// TwinCAT 3 PLC project SIM_1
// ProgramVersion: 3.1.4026.25
// libraries:
//   OC_Core, * (Open Commissioning)
//   OC_EtherCAT, * (Open Commissioning)
//   Tc2_Math, * (Beckhoff Automation GmbH)
//   Tc2_Standard, * (Beckhoff Automation GmbH)
//   Tc2_System, * (Beckhoff Automation GmbH)
//   Tc2_Utilities, * (Beckhoff Automation GmbH)
//   Tc3_Module, * (Beckhoff Automation GmbH)
// project tree:
//   Hil/EtherCAT_1_SIM/ GVL_EtherCAT_1_SIM.TcGVL, PRG_EtherCAT_1_SIM.TcPOU
//   Library/ FB_Camera.TcPOU (not stored)
//   FG_01/ FG_01.TcPOU
//   FG_02/ FG_02.TcPOU
//   FG_03/ FG_03.TcPOU
//   FG_04/ FG_04.TcPOU
//   FG_05/ FG_05.TcPOU
//   FG_System/ FG_System.TcPOU
//   FG_Transport/ FG_Transport.TcPOU
//   / MAIN.TcPOU, PlcTask.TcTTO (not stored)
// real-time tasks:
//   TASK PlcTask_SIM: cycle T#1ms, priority 4, ADS port 350
//   TASK PlcTask_PLC: cycle T#10ms, priority 20, ADS port 351
// I/O:
//   DEVICE EtherCAT_1_SIM, AmsNetId 169.254.215.222.4.1
//     FG_System_EK1100 // EK1100-0000-0018
//     FG_System_Panel_EL1809_1 // EL1809-0000-0018
//     FG_System_Panel_EL2809_1 // EL2809-0000-0018
//     FG_System_Door_EL1809_1 // EL1809-0000-0018
//     FG_System_Door_EL2008_1 // EL2008-0000-0018
//     FG_Transport_EK1100 // EK1100-0000-0018
//     FG_Transport_Index_EL1809_1 // EL1809-0000-0018
//     FG_Transport_Index_EL1809_2 // EL1809-0000-0018
//     FG_Transport_Stopper_EL1809_1 // EL1809-0000-0018
//     FG_Transport_Lift_EL1809_1 // EL1809-0000-0018
//     FG_Transport_Drive_EL1008_1 // EL1008-0000-0018
//     FG_Transport_Index_EL2809_1 // EL2809-0000-0018
//     FG_Transport_Stopper_EL2008_1 // EL2008-0000-0018
//     FG_Transport_Lift_EL2008_1 // EL2008-0000-0018
//     FG_Transport_Drive_EL2008_1 // EL2008-0000-0018
//     FG_01_EK1100 // EK1100-0000-0018
//     FG_01_EL1008_1 // EL1008-0000-0018
//     FG_01_EL1008_2 // EL1008-0000-0018
//     FG_01_EL2008_1 // EL2008-0000-0018
//     FG_01_EL1859_1 // EL1859-0000-0018
//     FG_01_EL1859_2 // EL1859-0000-0018
//     FG_02_EK1100 // EK1100-0000-0018
//     FG_02_EL1859_1 // EL1859-0000-0018
//     FG_03_EK1100 // EK1100-0000-0018
//     FG_03_EL1809_1 // EL1809-0000-0018
//     FG_03_EL2809_1 // EL2809-0000-0018
//     FG_04_EK1100 // EK1100-0000-0018
//     FG_04_EL1008_1 // EL1008-0000-0018
//     FG_04_EL2008_1 // EL2008-0000-0018
//     FG_05_EK1100 // EK1100-0000-0018
//     FG_05_EL1809_1 // EL1809-0000-0018
//     FG_05_EL2809_1 // EL2809-0000-0018
//     FG_05_EL1859_1 // EL1859-0000-0018
//     FG_05_EL1859_2 // EL1859-0000-0018
//   DEVICE EtherCAT_1, AmsNetId 169.254.215.222.3.1
//     FG_System_EK1100 [EK1100 EtherCAT Coupler (2A E-Bus)]
//       FG_System_Panel_EL1809_1 [EL1809 16Ch. Dig. Input 24V, 3ms]
//       FG_System_Panel_EL2809_1 [EL2809 16Ch. Dig. Output 24V, 0.5A]
//       FG_System_Door_EL1809_1 [EL1809 16Ch. Dig. Input 24V, 3ms]
//       FG_System_Door_EL2008_1 [EL2008 8Ch. Dig. Output 24V, 0.5A]
//     FG_Transport_EK1100 [EK1100 EtherCAT Coupler (2A E-Bus)]
//       FG_Transport_Index_EL1809_1 [EL1809 16Ch. Dig. Input 24V, 3ms]
//       FG_Transport_Index_EL1809_2 [EL1809 16Ch. Dig. Input 24V, 3ms]
//       FG_Transport_Stopper_EL1809_1 [EL1809 16Ch. Dig. Input 24V, 3ms]
//       FG_Transport_Lift_EL1809_1 [EL1809 16Ch. Dig. Input 24V, 3ms]
//       FG_Transport_Drive_EL1008_1 [EL1008 8Ch. Dig. Input 24V, 3ms]
//       FG_Transport_Index_EL2809_1 [EL2809 16Ch. Dig. Output 24V, 0.5A]
//       FG_Transport_Stopper_EL2008_1 [EL2008 8Ch. Dig. Output 24V, 0.5A]
//       FG_Transport_Lift_EL2008_1 [EL2008 8Ch. Dig. Output 24V, 0.5A]
//       FG_Transport_Drive_EL2008_1 [EL2008 8Ch. Dig. Output 24V, 0.5A]
//     FG_01_EK1100 [EK1100 EtherCAT Coupler (2A E-Bus)]
//       FG_01_EL1008_1 [EL1008 8Ch. Dig. Input 24V, 3ms]
//       FG_01_EL1008_2 [EL1008 8Ch. Dig. Input 24V, 3ms]
//       FG_01_EL2008_1 [EL2008 8Ch. Dig. Output 24V, 0.5A]
//       FG_01_EL1859_1 [EL1859 8Ch. Dig. Input 24V, 3ms, 8Ch. Dig. Output 24V, 0.5A]
//       FG_01_EL1859_2 [EL1859 8Ch. Dig. Input 24V, 3ms, 8Ch. Dig. Output 24V, 0.5A]
//     FG_02_EK1100 [EK1100 EtherCAT Coupler (2A E-Bus)]
//       FG_02_EL1859_1 [EL1859 8Ch. Dig. Input 24V, 3ms, 8Ch. Dig. Output 24V, 0.5A]
//     FG_03_EK1100 [EK1100 EtherCAT Coupler (2A E-Bus)]
//       FG_03_EL1809_1 [EL1809 16Ch. Dig. Input 24V, 3ms]
//       FG_03_EL2809_1 [EL2809 16Ch. Dig. Output 24V, 0.5A]
//     FG_04_EK1100 [EK1100 EtherCAT Coupler (2A E-Bus)]
//       FG_04_EL1008_1 [EL1008 8Ch. Dig. Input 24V, 3ms]
//       FG_04_EL2008_1 [EL2008 8Ch. Dig. Output 24V, 0.5A]
//     FG_05_EK1100 [EK1100 EtherCAT Coupler (2A E-Bus)]
//       FG_05_EL1809_1 [EL1809 16Ch. Dig. Input 24V, 3ms]
//       FG_05_EL2809_1 [EL2809 16Ch. Dig. Output 24V, 0.5A]
//       FG_05_EL1859_1 [EL1859 8Ch. Dig. Input 24V, 3ms, 8Ch. Dig. Output 24V, 0.5A]
//       FG_05_EL1859_2 [EL1859 8Ch. Dig. Input 24V, 3ms, 8Ch. Dig. Output 24V, 0.5A]
// variable links:
//   PLC_1/PLC_1 Instance <-> EtherCAT_1/FG_01_EK1100/FG_01_EL1008_1
//     PlcTask Inputs/MAIN.Machine.FG_01.Y_Gripper.ExtendedSensor <-> Channel 2/Input
//     PlcTask Inputs/MAIN.Machine.FG_01.Y_Gripper.RetractedSensor <-> Channel 1/Input
//     PlcTask Inputs/MAIN.Machine.FG_01.Y_Platform.ExtendedSensor <-> Channel 4/Input
//     PlcTask Inputs/MAIN.Machine.FG_01.Y_Platform.RetractedSensor <-> Channel 3/Input
//     PlcTask Inputs/MAIN.Machine.FG_01.Y_ReaderWindow.ExtendedSensor <-> Channel 6/Input
//     PlcTask Inputs/MAIN.Machine.FG_01.Y_ReaderWindow.RetractedSensor <-> Channel 5/Input
//   PLC_1/PLC_1 Instance <-> EtherCAT_1/FG_01_EK1100/FG_01_EL1008_2
//     PlcTask Inputs/MAIN.Machine.FG_01.B_SafetyGate1.HardwareInput <-> Channel 5/Input
//     PlcTask Inputs/MAIN.Machine.FG_01.B_SafetyGate2.HardwareInput <-> Channel 6/Input
//     PlcTask Inputs/MAIN.Machine.FG_01.Y_Gate1.ExtendedSensor <-> Channel 2/Input
//     PlcTask Inputs/MAIN.Machine.FG_01.Y_Gate2.ExtendedSensor <-> Channel 4/Input
//     PlcTask Inputs/MAIN.Machine.FG_01.Y_Gate1.RetractedSensor <-> Channel 1/Input
//     PlcTask Inputs/MAIN.Machine.FG_01.Y_Gate2.RetractedSensor <-> Channel 3/Input
//   PLC_1/PLC_1 Instance <-> EtherCAT_1/FG_01_EK1100/FG_01_EL1859_1
//     PlcTask Inputs/MAIN.Machine.FG_01.P_Camera.InputData <-> Channel 1/Input
//     PlcTask Inputs/MAIN.Machine.FG_01.P_Camera.InputData @bit 1 <-> Channel 2/Input
//     PlcTask Inputs/MAIN.Machine.FG_01.P_Camera.InputData @bit 2 <-> Channel 3/Input
//     PlcTask Inputs/MAIN.Machine.FG_01.P_Camera.InputData @bit 3 <-> Channel 4/Input
//     PlcTask Inputs/MAIN.Machine.FG_01.P_Camera.InputData @bit 4 <-> Channel 5/Input
//     PlcTask Inputs/MAIN.Machine.FG_01.P_Camera.InputData @bit 5 <-> Channel 6/Input
//     PlcTask Inputs/MAIN.Machine.FG_01.P_Camera.InputData @bit 6 <-> Channel 7/Input
//     PlcTask Inputs/MAIN.Machine.FG_01.P_Camera.InputData @bit 7 <-> Channel 8/Input
//     PlcTask Outputs/MAIN.Machine.FG_01.P_Camera.OutputData @bit 1 <-> Channel 10/Output
//     PlcTask Outputs/MAIN.Machine.FG_01.P_Camera.OutputData @bit 2 <-> Channel 11/Output
//     PlcTask Outputs/MAIN.Machine.FG_01.P_Camera.OutputData @bit 3 <-> Channel 12/Output
//     PlcTask Outputs/MAIN.Machine.FG_01.P_Camera.OutputData @bit 4 <-> Channel 13/Output
//     PlcTask Outputs/MAIN.Machine.FG_01.P_Camera.OutputData @bit 5 <-> Channel 14/Output
//     PlcTask Outputs/MAIN.Machine.FG_01.P_Camera.OutputData @bit 6 <-> Channel 15/Output
//     PlcTask Outputs/MAIN.Machine.FG_01.P_Camera.OutputData @bit 7 <-> Channel 16/Output
//     PlcTask Outputs/MAIN.Machine.FG_01.P_Camera.OutputData <-> Channel 9/Output
//   PLC_1/PLC_1 Instance <-> EtherCAT_1/FG_01_EK1100/FG_01_EL1859_2
//     PlcTask Inputs/MAIN.Machine.FG_01.Y_LaserMark.InputData <-> Channel 1/Input
//     PlcTask Inputs/MAIN.Machine.FG_01.Y_LaserMark.InputData @bit 1 <-> Channel 2/Input
//     PlcTask Inputs/MAIN.Machine.FG_01.Y_LaserMark.InputData @bit 2 <-> Channel 3/Input
//     PlcTask Inputs/MAIN.Machine.FG_01.Y_LaserMark.InputData @bit 3 <-> Channel 4/Input
//     PlcTask Inputs/MAIN.Machine.FG_01.Y_LaserMark.InputData @bit 4 <-> Channel 5/Input
//     PlcTask Inputs/MAIN.Machine.FG_01.Y_LaserMark.InputData @bit 5 <-> Channel 6/Input
//     PlcTask Inputs/MAIN.Machine.FG_01.Y_LaserMark.InputData @bit 6 <-> Channel 7/Input
//     PlcTask Inputs/MAIN.Machine.FG_01.Y_LaserMark.InputData @bit 7 <-> Channel 8/Input
//     PlcTask Outputs/MAIN.Machine.FG_01.Y_LaserMark.OutputData @bit 1 <-> Channel 10/Output
//     PlcTask Outputs/MAIN.Machine.FG_01.Y_LaserMark.OutputData @bit 2 <-> Channel 11/Output
//     PlcTask Outputs/MAIN.Machine.FG_01.Y_LaserMark.OutputData @bit 3 <-> Channel 12/Output
//     PlcTask Outputs/MAIN.Machine.FG_01.Y_LaserMark.OutputData @bit 4 <-> Channel 13/Output
//     PlcTask Outputs/MAIN.Machine.FG_01.Y_LaserMark.OutputData @bit 5 <-> Channel 14/Output
//     PlcTask Outputs/MAIN.Machine.FG_01.Y_LaserMark.OutputData @bit 6 <-> Channel 15/Output
//     PlcTask Outputs/MAIN.Machine.FG_01.Y_LaserMark.OutputData @bit 7 <-> Channel 16/Output
//     PlcTask Outputs/MAIN.Machine.FG_01.Y_LaserMark.OutputData <-> Channel 9/Output
//   PLC_1/PLC_1 Instance <-> EtherCAT_1/FG_01_EK1100/FG_01_EL2008_1
//     PlcTask Outputs/MAIN.Machine.FG_01.Y_Gate1._ExtendOutput <-> Channel 7/Output
//     PlcTask Outputs/MAIN.Machine.FG_01.Y_Gate2._ExtendOutput <-> Channel 8/Output
//     PlcTask Outputs/MAIN.Machine.FG_01.Y_Gripper._ExtendOutput <-> Channel 1/Output
//     PlcTask Outputs/MAIN.Machine.FG_01.Y_Gripper._RetractOutput <-> Channel 5/Output
//     PlcTask Outputs/MAIN.Machine.FG_01.Y_Platform._ExtendOutput <-> Channel 2/Output
//     PlcTask Outputs/MAIN.Machine.FG_01.Y_Platform._RetractOutput <-> Channel 3/Output
//     PlcTask Outputs/MAIN.Machine.FG_01.Y_ReaderWindow._ExtendOutput <-> Channel 4/Output
//     PlcTask Outputs/MAIN.Machine.FG_01.Y_ReaderWindow._RetractOutput <-> Channel 6/Output
//   PLC_1/PLC_1 Instance <-> EtherCAT_1/FG_02_EK1100/FG_02_EL1859_1
//     PlcTask Inputs/MAIN.Machine.FG_02.P_Camera.InputData <-> Channel 1/Input
//     PlcTask Inputs/MAIN.Machine.FG_02.P_Camera.InputData @bit 1 <-> Channel 2/Input
//     PlcTask Inputs/MAIN.Machine.FG_02.P_Camera.InputData @bit 2 <-> Channel 3/Input
//     PlcTask Inputs/MAIN.Machine.FG_02.P_Camera.InputData @bit 3 <-> Channel 4/Input
//     PlcTask Inputs/MAIN.Machine.FG_02.P_Camera.InputData @bit 4 <-> Channel 5/Input
//     PlcTask Inputs/MAIN.Machine.FG_02.P_Camera.InputData @bit 5 <-> Channel 6/Input
//     PlcTask Inputs/MAIN.Machine.FG_02.P_Camera.InputData @bit 6 <-> Channel 7/Input
//     PlcTask Inputs/MAIN.Machine.FG_02.P_Camera.InputData @bit 7 <-> Channel 8/Input
//     PlcTask Outputs/MAIN.Machine.FG_02.P_Camera.OutputData @bit 1 <-> Channel 10/Output
//     PlcTask Outputs/MAIN.Machine.FG_02.P_Camera.OutputData @bit 2 <-> Channel 11/Output
//     PlcTask Outputs/MAIN.Machine.FG_02.P_Camera.OutputData @bit 3 <-> Channel 12/Output
//     PlcTask Outputs/MAIN.Machine.FG_02.P_Camera.OutputData @bit 4 <-> Channel 13/Output
//     PlcTask Outputs/MAIN.Machine.FG_02.P_Camera.OutputData @bit 5 <-> Channel 14/Output
//     PlcTask Outputs/MAIN.Machine.FG_02.P_Camera.OutputData @bit 6 <-> Channel 15/Output
//     PlcTask Outputs/MAIN.Machine.FG_02.P_Camera.OutputData @bit 7 <-> Channel 16/Output
//     PlcTask Outputs/MAIN.Machine.FG_02.P_Camera.OutputData <-> Channel 9/Output
//   PLC_1/PLC_1 Instance <-> EtherCAT_1/FG_03_EK1100/FG_03_EL1809_1
//     PlcTask Inputs/MAIN.Machine.FG_03.B_Detect1.HardwareInput <-> Channel 15/Input
//     PlcTask Inputs/MAIN.Machine.FG_03.B_Detect2.HardwareInput <-> Channel 16/Input
//     PlcTask Inputs/MAIN.Machine.FG_03.Y_AxisR1.ExtendedSensor <-> Channel 5/Input
//     PlcTask Inputs/MAIN.Machine.FG_03.Y_AxisR1.RetractedSensor <-> Channel 6/Input
//     PlcTask Inputs/MAIN.Machine.FG_03.Y_AxisX1.ExtendedSensor <-> Channel 1/Input
//     PlcTask Inputs/MAIN.Machine.FG_03.Y_AxisX2.ExtendedSensor <-> Channel 9/Input
//     PlcTask Inputs/MAIN.Machine.FG_03.Y_AxisX1.RetractedSensor <-> Channel 2/Input
//     PlcTask Inputs/MAIN.Machine.FG_03.Y_AxisX2.RetractedSensor <-> Channel 10/Input
//     PlcTask Inputs/MAIN.Machine.FG_03.Y_AxisY1.ExtendedSensor <-> Channel 3/Input
//     PlcTask Inputs/MAIN.Machine.FG_03.Y_AxisY2.ExtendedSensor <-> Channel 11/Input
//     PlcTask Inputs/MAIN.Machine.FG_03.Y_AxisY1.RetractedSensor <-> Channel 4/Input
//     PlcTask Inputs/MAIN.Machine.FG_03.Y_AxisY2.RetractedSensor <-> Channel 12/Input
//     PlcTask Inputs/MAIN.Machine.FG_03.Y_Gripper1.ExtendedSensor <-> Channel 7/Input
//     PlcTask Inputs/MAIN.Machine.FG_03.Y_Gripper2.ExtendedSensor <-> Channel 13/Input
//     PlcTask Inputs/MAIN.Machine.FG_03.Y_Gripper1.RetractedSensor <-> Channel 8/Input
//     PlcTask Inputs/MAIN.Machine.FG_03.Y_Gripper2.RetractedSensor <-> Channel 14/Input
//   PLC_1/PLC_1 Instance <-> EtherCAT_1/FG_03_EK1100/FG_03_EL2809_1
//     PlcTask Outputs/MAIN.Machine.FG_03.Y_AxisR1._ExtendOutput <-> Channel 5/Output
//     PlcTask Outputs/MAIN.Machine.FG_03.Y_AxisR1._RetractOutput <-> Channel 6/Output
//     PlcTask Outputs/MAIN.Machine.FG_03.Y_AxisX1._ExtendOutput <-> Channel 1/Output
//     PlcTask Outputs/MAIN.Machine.FG_03.Y_AxisX2._ExtendOutput <-> Channel 9/Output
//     PlcTask Outputs/MAIN.Machine.FG_03.Y_AxisX1._RetractOutput <-> Channel 2/Output
//     PlcTask Outputs/MAIN.Machine.FG_03.Y_AxisX2._RetractOutput <-> Channel 10/Output
//     PlcTask Outputs/MAIN.Machine.FG_03.Y_AxisY1._ExtendOutput <-> Channel 3/Output
//     PlcTask Outputs/MAIN.Machine.FG_03.Y_AxisY2._ExtendOutput <-> Channel 11/Output
//     PlcTask Outputs/MAIN.Machine.FG_03.Y_AxisY1._RetractOutput <-> Channel 4/Output
//     PlcTask Outputs/MAIN.Machine.FG_03.Y_AxisY2._RetractOutput <-> Channel 12/Output
//     PlcTask Outputs/MAIN.Machine.FG_03.Y_Gripper1._ExtendOutput <-> Channel 7/Output
//     PlcTask Outputs/MAIN.Machine.FG_03.Y_Gripper2._ExtendOutput <-> Channel 13/Output
//     PlcTask Outputs/MAIN.Machine.FG_03.Y_Gripper1._RetractOutput <-> Channel 8/Output
//     PlcTask Outputs/MAIN.Machine.FG_03.Y_Gripper2._RetractOutput <-> Channel 14/Output
//   PLC_1/PLC_1 Instance <-> EtherCAT_1/FG_04_EK1100/FG_04_EL1008_1
//     PlcTask Inputs/MAIN.Machine.FG_04.B_NIO.HardwareInput <-> Channel 3/Input
//     PlcTask Inputs/MAIN.Machine.FG_04.Y_AxisZ.ExtendedSensor <-> Channel 1/Input
//     PlcTask Inputs/MAIN.Machine.FG_04.Y_AxisZ.RetractedSensor <-> Channel 2/Input
//   PLC_1/PLC_1 Instance <-> EtherCAT_1/FG_04_EK1100/FG_04_EL2008_1
//     PlcTask Outputs/MAIN.Machine.FG_04.Y_AxisZ._ExtendOutput <-> Channel 1/Output
//     PlcTask Outputs/MAIN.Machine.FG_04.Y_AxisZ._RetractOutput <-> Channel 2/Output
//   PLC_1/PLC_1 Instance <-> EtherCAT_1/FG_05_EK1100/FG_05_EL1809_1
//     PlcTask Inputs/MAIN.Machine.FG_05.B_Detect.HardwareInput <-> Channel 14/Input
//     PlcTask Inputs/MAIN.Machine.FG_05.B_Part.HardwareInput <-> Channel 13/Input
//     PlcTask Inputs/MAIN.Machine.FG_05.Y_AxisR.ExtendedSensor <-> Channel 7/Input
//     PlcTask Inputs/MAIN.Machine.FG_05.Y_AxisR.RetractedSensor <-> Channel 8/Input
//     PlcTask Inputs/MAIN.Machine.FG_05.Y_AxisX.ExtendedSensor <-> Channel 1/Input
//     PlcTask Inputs/MAIN.Machine.FG_05.Y_AxisX.RetractedSensor <-> Channel 2/Input
//     PlcTask Inputs/MAIN.Machine.FG_05.Y_AxisZ1.ExtendedSensor <-> Channel 3/Input
//     PlcTask Inputs/MAIN.Machine.FG_05.Y_AxisZ2.ExtendedSensor <-> Channel 5/Input
//     PlcTask Inputs/MAIN.Machine.FG_05.Y_AxisZ1.RetractedSensor <-> Channel 4/Input
//     PlcTask Inputs/MAIN.Machine.FG_05.Y_AxisZ2.RetractedSensor <-> Channel 6/Input
//     PlcTask Inputs/MAIN.Machine.FG_05.Y_CapsSourceStopper.ExtendedSensor <-> Channel 11/Input
//     PlcTask Inputs/MAIN.Machine.FG_05.Y_CapsSourceStopper.RetractedSensor <-> Channel 12/Input
//     PlcTask Inputs/MAIN.Machine.FG_05.Y_Gripper.ExtendedSensor <-> Channel 9/Input
//     PlcTask Inputs/MAIN.Machine.FG_05.Y_Gripper.RetractedSensor <-> Channel 10/Input
//   PLC_1/PLC_1 Instance <-> EtherCAT_1/FG_05_EK1100/FG_05_EL1859_1
//     PlcTask Inputs/MAIN.Machine.FG_05.Y_CapsSource.InputData <-> Channel 1/Input
//     PlcTask Inputs/MAIN.Machine.FG_05.Y_CapsSource.InputData @bit 1 <-> Channel 2/Input
//     PlcTask Inputs/MAIN.Machine.FG_05.Y_CapsSource.InputData @bit 2 <-> Channel 3/Input
//     PlcTask Inputs/MAIN.Machine.FG_05.Y_CapsSource.InputData @bit 3 <-> Channel 4/Input
//     PlcTask Inputs/MAIN.Machine.FG_05.Y_CapsSource.InputData @bit 4 <-> Channel 5/Input
//     PlcTask Inputs/MAIN.Machine.FG_05.Y_CapsSource.InputData @bit 5 <-> Channel 6/Input
//     PlcTask Inputs/MAIN.Machine.FG_05.Y_CapsSource.InputData @bit 6 <-> Channel 7/Input
//     PlcTask Inputs/MAIN.Machine.FG_05.Y_CapsSource.InputData @bit 7 <-> Channel 8/Input
//     PlcTask Outputs/MAIN.Machine.FG_05.Y_CapsSource.OutputData @bit 1 <-> Channel 10/Output
//     PlcTask Outputs/MAIN.Machine.FG_05.Y_CapsSource.OutputData @bit 2 <-> Channel 11/Output
//     PlcTask Outputs/MAIN.Machine.FG_05.Y_CapsSource.OutputData @bit 3 <-> Channel 12/Output
//     PlcTask Outputs/MAIN.Machine.FG_05.Y_CapsSource.OutputData @bit 4 <-> Channel 13/Output
//     PlcTask Outputs/MAIN.Machine.FG_05.Y_CapsSource.OutputData @bit 5 <-> Channel 14/Output
//     PlcTask Outputs/MAIN.Machine.FG_05.Y_CapsSource.OutputData @bit 6 <-> Channel 15/Output
//     PlcTask Outputs/MAIN.Machine.FG_05.Y_CapsSource.OutputData @bit 7 <-> Channel 16/Output
//     PlcTask Outputs/MAIN.Machine.FG_05.Y_CapsSource.OutputData <-> Channel 9/Output
//   PLC_1/PLC_1 Instance <-> EtherCAT_1/FG_05_EK1100/FG_05_EL1859_2
//     PlcTask Inputs/MAIN.Machine.FG_05.P_Camera.InputData <-> Channel 1/Input
//     PlcTask Inputs/MAIN.Machine.FG_05.P_Camera.InputData @bit 1 <-> Channel 2/Input
//     PlcTask Inputs/MAIN.Machine.FG_05.P_Camera.InputData @bit 2 <-> Channel 3/Input
//     PlcTask Inputs/MAIN.Machine.FG_05.P_Camera.InputData @bit 3 <-> Channel 4/Input
//     PlcTask Inputs/MAIN.Machine.FG_05.P_Camera.InputData @bit 4 <-> Channel 5/Input
//     PlcTask Inputs/MAIN.Machine.FG_05.P_Camera.InputData @bit 5 <-> Channel 6/Input
//     PlcTask Inputs/MAIN.Machine.FG_05.P_Camera.InputData @bit 6 <-> Channel 7/Input
//     PlcTask Inputs/MAIN.Machine.FG_05.P_Camera.InputData @bit 7 <-> Channel 8/Input
//     PlcTask Outputs/MAIN.Machine.FG_05.P_Camera.OutputData @bit 1 <-> Channel 10/Output
//     PlcTask Outputs/MAIN.Machine.FG_05.P_Camera.OutputData @bit 2 <-> Channel 11/Output
//     PlcTask Outputs/MAIN.Machine.FG_05.P_Camera.OutputData @bit 3 <-> Channel 12/Output
//     PlcTask Outputs/MAIN.Machine.FG_05.P_Camera.OutputData @bit 4 <-> Channel 13/Output
//     PlcTask Outputs/MAIN.Machine.FG_05.P_Camera.OutputData @bit 5 <-> Channel 14/Output
//     PlcTask Outputs/MAIN.Machine.FG_05.P_Camera.OutputData @bit 6 <-> Channel 15/Output
//     PlcTask Outputs/MAIN.Machine.FG_05.P_Camera.OutputData @bit 7 <-> Channel 16/Output
//     PlcTask Outputs/MAIN.Machine.FG_05.P_Camera.OutputData <-> Channel 9/Output
//   PLC_1/PLC_1 Instance <-> EtherCAT_1/FG_05_EK1100/FG_05_EL2809_1
//     PlcTask Outputs/MAIN.Machine.FG_05.Y_AxisR._ExtendOutput <-> Channel 7/Output
//     PlcTask Outputs/MAIN.Machine.FG_05.Y_AxisR._RetractOutput <-> Channel 8/Output
//     PlcTask Outputs/MAIN.Machine.FG_05.Y_AxisX._ExtendOutput <-> Channel 1/Output
//     PlcTask Outputs/MAIN.Machine.FG_05.Y_AxisX._RetractOutput <-> Channel 2/Output
//     PlcTask Outputs/MAIN.Machine.FG_05.Y_AxisZ1._ExtendOutput <-> Channel 3/Output
//     PlcTask Outputs/MAIN.Machine.FG_05.Y_AxisZ2._ExtendOutput <-> Channel 5/Output
//     PlcTask Outputs/MAIN.Machine.FG_05.Y_AxisZ1._RetractOutput <-> Channel 4/Output
//     PlcTask Outputs/MAIN.Machine.FG_05.Y_AxisZ2._RetractOutput <-> Channel 6/Output
//     PlcTask Outputs/MAIN.Machine.FG_05.Y_CapsSourceStopper._ExtendOutput <-> Channel 11/Output
//     PlcTask Outputs/MAIN.Machine.FG_05.Y_CapsSourceStopper._RetractOutput <-> Channel 12/Output
//     PlcTask Outputs/MAIN.Machine.FG_05.Y_Gripper._ExtendOutput <-> Channel 9/Output
//     PlcTask Outputs/MAIN.Machine.FG_05.Y_Gripper._RetractOutput <-> Channel 10/Output
//   PLC_1/PLC_1 Instance <-> EtherCAT_1/FG_System_EK1100/FG_System_Door_EL1809_1
//     PlcTask Inputs/MAIN.Machine.FG_System.B_SafetyDoor11.ClosedSensor <-> Channel 1/Input
//     PlcTask Inputs/MAIN.Machine.FG_System.B_SafetyDoor12.ClosedSensor <-> Channel 3/Input
//     PlcTask Inputs/MAIN.Machine.FG_System.B_SafetyDoor13.ClosedSensor <-> Channel 5/Input
//     PlcTask Inputs/MAIN.Machine.FG_System.B_SafetyDoor21.ClosedSensor <-> Channel 7/Input
//     PlcTask Inputs/MAIN.Machine.FG_System.B_SafetyDoor22.ClosedSensor <-> Channel 9/Input
//     PlcTask Inputs/MAIN.Machine.FG_System.B_SafetyDoor23.ClosedSensor <-> Channel 11/Input
//     PlcTask Inputs/MAIN.Machine.FG_System.B_SafetyDoor11.LockedSensor <-> Channel 2/Input
//     PlcTask Inputs/MAIN.Machine.FG_System.B_SafetyDoor12.LockedSensor <-> Channel 4/Input
//     PlcTask Inputs/MAIN.Machine.FG_System.B_SafetyDoor13.LockedSensor <-> Channel 6/Input
//     PlcTask Inputs/MAIN.Machine.FG_System.B_SafetyDoor21.LockedSensor <-> Channel 8/Input
//     PlcTask Inputs/MAIN.Machine.FG_System.B_SafetyDoor22.LockedSensor <-> Channel 10/Input
//     PlcTask Inputs/MAIN.Machine.FG_System.B_SafetyDoor23.LockedSensor <-> Channel 12/Input
//   PLC_1/PLC_1 Instance <-> EtherCAT_1/FG_System_EK1100/FG_System_Door_EL2008_1
//     PlcTask Outputs/MAIN.Machine.FG_System.B_SafetyDoor11.LockOutput <-> Channel 1/Output
//     PlcTask Outputs/MAIN.Machine.FG_System.B_SafetyDoor12.LockOutput <-> Channel 2/Output
//     PlcTask Outputs/MAIN.Machine.FG_System.B_SafetyDoor13.LockOutput <-> Channel 3/Output
//     PlcTask Outputs/MAIN.Machine.FG_System.B_SafetyDoor21.LockOutput <-> Channel 4/Output
//     PlcTask Outputs/MAIN.Machine.FG_System.B_SafetyDoor22.LockOutput <-> Channel 5/Output
//     PlcTask Outputs/MAIN.Machine.FG_System.B_SafetyDoor23.LockOutput <-> Channel 6/Output
//   PLC_1/PLC_1 Instance <-> EtherCAT_1/FG_System_EK1100/FG_System_Panel_EL1809_1
//     PlcTask Inputs/MAIN.ControlSource_Panel.AbortPressed <-> Channel 5/Input
//     PlcTask Inputs/MAIN.ControlSource_Panel.ClearPressed <-> Channel 4/Input
//     PlcTask Inputs/MAIN.ControlSource_Panel.MainPMLControl_Simplified.ResetPressed <-> Channel 2/Input
//     PlcTask Inputs/MAIN.ControlSource_Panel.MainPMLControl_Simplified.StartPressed <-> Channel 1/Input
//     PlcTask Inputs/MAIN.ControlSource_Panel.MainPMLControl_Simplified.StopPressed <-> Channel 3/Input
//     PlcTask Inputs/MAIN.ControlSource_Panel.MaintenancePressed <-> Channel 7/Input
//     PlcTask Inputs/MAIN.ControlSource_Panel.ManualPressed <-> Channel 8/Input
//     PlcTask Inputs/MAIN.ControlSource_Panel.ProductionPressed <-> Channel 6/Input
//     PlcTask Inputs/MAIN.Machine.FG_System.SS_EStop1.HardwareInput <-> Channel 9/Input
//     PlcTask Inputs/MAIN.Machine.FG_System.SS_EStop2.HardwareInput <-> Channel 10/Input
//   PLC_1/PLC_1 Instance <-> EtherCAT_1/FG_System_EK1100/FG_System_Panel_EL2809_1
//     PlcTask Outputs/MAIN.ControlSource_Panel.LampAbort <-> Channel 5/Output
//     PlcTask Outputs/MAIN.ControlSource_Panel.LampClear <-> Channel 4/Output
//     PlcTask Outputs/MAIN.ControlSource_Panel.LampMaintenance <-> Channel 7/Output
//     PlcTask Outputs/MAIN.ControlSource_Panel.LampManual <-> Channel 8/Output
//     PlcTask Outputs/MAIN.ControlSource_Panel.LampProduction <-> Channel 6/Output
//     PlcTask Outputs/MAIN.ControlSource_Panel.LampReset <-> Channel 2/Output
//     PlcTask Outputs/MAIN.ControlSource_Panel.LampStart <-> Channel 1/Output
//     PlcTask Outputs/MAIN.ControlSource_Panel.LampStop <-> Channel 3/Output
//     PlcTask Outputs/MAIN.Machine.FG_System.H_SignalTower.Blue <-> Channel 11/Output
//     PlcTask Outputs/MAIN.Machine.FG_System.H_SignalTower.Green <-> Channel 12/Output
//     PlcTask Outputs/MAIN.Machine.FG_System.H_SignalTower.Red <-> Channel 9/Output
//     PlcTask Outputs/MAIN.Machine.FG_System.H_SignalTower.Yellow <-> Channel 10/Output
//     PlcTask Outputs/MAIN.Machine.FG_System.SS_EStop1.LampOutput <-> Channel 13/Output
//     PlcTask Outputs/MAIN.Machine.FG_System.SS_EStop2.LampOutput <-> Channel 14/Output
//   PLC_1/PLC_1 Instance <-> EtherCAT_1/FG_Transport_EK1100/FG_Transport_Drive_EL1008_1
//     PlcTask Inputs/MAIN.Machine.FG_Transport.Transport01._DriveActive <-> Channel 1/Input
//     PlcTask Inputs/MAIN.Machine.FG_Transport.Transport02._DriveActive <-> Channel 2/Input
//   PLC_1/PLC_1 Instance <-> EtherCAT_1/FG_Transport_EK1100/FG_Transport_Drive_EL2008_1
//     PlcTask Outputs/MAIN.Machine.FG_Transport.Transport01._Backward <-> Channel 1/Output
//     PlcTask Outputs/MAIN.Machine.FG_Transport.Transport02._Backward <-> Channel 3/Output
//     PlcTask Outputs/MAIN.Machine.FG_Transport.Transport01._Forward <-> Channel 2/Output
//     PlcTask Outputs/MAIN.Machine.FG_Transport.Transport02._Forward <-> Channel 4/Output
//   PLC_1/PLC_1 Instance <-> EtherCAT_1/FG_Transport_EK1100/FG_Transport_Index_EL1809_1
//     PlcTask Inputs/MAIN.Machine.FG_Transport.Index01.B_Detect.HardwareInput <-> Channel 1/Input
//     PlcTask Inputs/MAIN.Machine.FG_Transport.Index02.B_Detect.HardwareInput <-> Channel 7/Input
//     PlcTask Inputs/MAIN.Machine.FG_Transport.Index03.B_Detect.HardwareInput <-> Channel 13/Input
//     PlcTask Inputs/MAIN.Machine.FG_Transport.Index01.B_Exit.HardwareInput <-> Channel 2/Input
//     PlcTask Inputs/MAIN.Machine.FG_Transport.Index02.B_Exit.HardwareInput <-> Channel 8/Input
//     PlcTask Inputs/MAIN.Machine.FG_Transport.Index03.B_Exit.HardwareInput <-> Channel 14/Input
//     PlcTask Inputs/MAIN.Machine.FG_Transport.Index01.Y_Lift.ExtendedSensor <-> Channel 4/Input
//     PlcTask Inputs/MAIN.Machine.FG_Transport.Index02.Y_Lift.ExtendedSensor <-> Channel 10/Input
//     PlcTask Inputs/MAIN.Machine.FG_Transport.Index03.Y_Lift.ExtendedSensor <-> Channel 16/Input
//     PlcTask Inputs/MAIN.Machine.FG_Transport.Index01.Y_Lift.RetractedSensor <-> Channel 3/Input
//     PlcTask Inputs/MAIN.Machine.FG_Transport.Index02.Y_Lift.RetractedSensor <-> Channel 9/Input
//     PlcTask Inputs/MAIN.Machine.FG_Transport.Index03.Y_Lift.RetractedSensor <-> Channel 15/Input
//     PlcTask Inputs/MAIN.Machine.FG_Transport.Index01.Y_Stopper.ExtendedSensor <-> Channel 6/Input
//     PlcTask Inputs/MAIN.Machine.FG_Transport.Index02.Y_Stopper.ExtendedSensor <-> Channel 12/Input
//     PlcTask Inputs/MAIN.Machine.FG_Transport.Index01.Y_Stopper.RetractedSensor <-> Channel 5/Input
//     PlcTask Inputs/MAIN.Machine.FG_Transport.Index02.Y_Stopper.RetractedSensor <-> Channel 11/Input
//   PLC_1/PLC_1 Instance <-> EtherCAT_1/FG_Transport_EK1100/FG_Transport_Index_EL1809_2
//     PlcTask Inputs/MAIN.Machine.FG_Transport.Index03.Y_Stopper.ExtendedSensor <-> Channel 2/Input
//     PlcTask Inputs/MAIN.Machine.FG_Transport.Index04.Y_Stopper.ExtendedSensor <-> Channel 8/Input
//     PlcTask Inputs/MAIN.Machine.FG_Transport.Index05.Y_Stopper.ExtendedSensor <-> Channel 14/Input
//     PlcTask Inputs/MAIN.Machine.FG_Transport.Index03.Y_Stopper.RetractedSensor <-> Channel 1/Input
//     PlcTask Inputs/MAIN.Machine.FG_Transport.Index04.Y_Stopper.RetractedSensor <-> Channel 7/Input
//     PlcTask Inputs/MAIN.Machine.FG_Transport.Index05.Y_Stopper.RetractedSensor <-> Channel 13/Input
//     PlcTask Inputs/MAIN.Machine.FG_Transport.Index04.B_Detect.HardwareInput <-> Channel 3/Input
//     PlcTask Inputs/MAIN.Machine.FG_Transport.Index05.B_Detect.HardwareInput <-> Channel 9/Input
//     PlcTask Inputs/MAIN.Machine.FG_Transport.Index04.B_Exit.HardwareInput <-> Channel 4/Input
//     PlcTask Inputs/MAIN.Machine.FG_Transport.Index05.B_Exit.HardwareInput <-> Channel 10/Input
//     PlcTask Inputs/MAIN.Machine.FG_Transport.Index04.Y_Lift.ExtendedSensor <-> Channel 6/Input
//     PlcTask Inputs/MAIN.Machine.FG_Transport.Index05.Y_Lift.ExtendedSensor <-> Channel 12/Input
//     PlcTask Inputs/MAIN.Machine.FG_Transport.Index04.Y_Lift.RetractedSensor <-> Channel 5/Input
//     PlcTask Inputs/MAIN.Machine.FG_Transport.Index05.Y_Lift.RetractedSensor <-> Channel 11/Input
//   PLC_1/PLC_1 Instance <-> EtherCAT_1/FG_Transport_EK1100/FG_Transport_Index_EL2809_1
//     PlcTask Outputs/MAIN.Machine.FG_Transport.Index01.Y_Lift._ExtendOutput <-> Channel 2/Output
//     PlcTask Outputs/MAIN.Machine.FG_Transport.Index02.Y_Lift._ExtendOutput <-> Channel 5/Output
//     PlcTask Outputs/MAIN.Machine.FG_Transport.Index03.Y_Lift._ExtendOutput <-> Channel 8/Output
//     PlcTask Outputs/MAIN.Machine.FG_Transport.Index04.Y_Lift._ExtendOutput <-> Channel 11/Output
//     PlcTask Outputs/MAIN.Machine.FG_Transport.Index05.Y_Lift._ExtendOutput <-> Channel 14/Output
//     PlcTask Outputs/MAIN.Machine.FG_Transport.Index01.Y_Lift._RetractOutput <-> Channel 1/Output
//     PlcTask Outputs/MAIN.Machine.FG_Transport.Index02.Y_Lift._RetractOutput <-> Channel 4/Output
//     PlcTask Outputs/MAIN.Machine.FG_Transport.Index03.Y_Lift._RetractOutput <-> Channel 7/Output
//     PlcTask Outputs/MAIN.Machine.FG_Transport.Index04.Y_Lift._RetractOutput <-> Channel 10/Output
//     PlcTask Outputs/MAIN.Machine.FG_Transport.Index05.Y_Lift._RetractOutput <-> Channel 13/Output
//     PlcTask Outputs/MAIN.Machine.FG_Transport.Index01.Y_Stopper._ExtendOutput <-> Channel 3/Output
//     PlcTask Outputs/MAIN.Machine.FG_Transport.Index02.Y_Stopper._ExtendOutput <-> Channel 6/Output
//     PlcTask Outputs/MAIN.Machine.FG_Transport.Index03.Y_Stopper._ExtendOutput <-> Channel 9/Output
//     PlcTask Outputs/MAIN.Machine.FG_Transport.Index04.Y_Stopper._ExtendOutput <-> Channel 12/Output
//     PlcTask Outputs/MAIN.Machine.FG_Transport.Index05.Y_Stopper._ExtendOutput <-> Channel 15/Output
//   PLC_1/PLC_1 Instance <-> EtherCAT_1/FG_Transport_EK1100/FG_Transport_Lift_EL1809_1
//     PlcTask Inputs/MAIN.Machine.FG_Transport.Lift01.B_Detect.HardwareInput <-> Channel 1/Input
//     PlcTask Inputs/MAIN.Machine.FG_Transport.Lift02.B_Detect.HardwareInput <-> Channel 6/Input
//     PlcTask Inputs/MAIN.Machine.FG_Transport.Lift01.B_Exit.HardwareInput <-> Channel 2/Input
//     PlcTask Inputs/MAIN.Machine.FG_Transport.Lift02.B_Exit.HardwareInput <-> Channel 7/Input
//     PlcTask Inputs/MAIN.Machine.FG_Transport.Lift01.M_Conveyor._DriveActive <-> Channel 5/Input
//     PlcTask Inputs/MAIN.Machine.FG_Transport.Lift02.M_Conveyor._DriveActive <-> Channel 10/Input
//     PlcTask Inputs/MAIN.Machine.FG_Transport.Lift01.Y_Lift.ExtendedSensor <-> Channel 4/Input
//     PlcTask Inputs/MAIN.Machine.FG_Transport.Lift02.Y_Lift.ExtendedSensor <-> Channel 9/Input
//     PlcTask Inputs/MAIN.Machine.FG_Transport.Lift01.Y_Lift.RetractedSensor <-> Channel 3/Input
//     PlcTask Inputs/MAIN.Machine.FG_Transport.Lift02.Y_Lift.RetractedSensor <-> Channel 8/Input
//   PLC_1/PLC_1 Instance <-> EtherCAT_1/FG_Transport_EK1100/FG_Transport_Lift_EL2008_1
//     PlcTask Outputs/MAIN.Machine.FG_Transport.Lift01.M_Conveyor._Backward <-> Channel 3/Output
//     PlcTask Outputs/MAIN.Machine.FG_Transport.Lift02.M_Conveyor._Backward <-> Channel 7/Output
//     PlcTask Outputs/MAIN.Machine.FG_Transport.Lift01.M_Conveyor._Forward <-> Channel 4/Output
//     PlcTask Outputs/MAIN.Machine.FG_Transport.Lift02.M_Conveyor._Forward <-> Channel 8/Output
//     PlcTask Outputs/MAIN.Machine.FG_Transport.Lift01.Y_Lift._ExtendOutput <-> Channel 2/Output
//     PlcTask Outputs/MAIN.Machine.FG_Transport.Lift02.Y_Lift._ExtendOutput <-> Channel 6/Output
//     PlcTask Outputs/MAIN.Machine.FG_Transport.Lift01.Y_Lift._RetractOutput <-> Channel 1/Output
//     PlcTask Outputs/MAIN.Machine.FG_Transport.Lift02.Y_Lift._RetractOutput <-> Channel 5/Output
//   PLC_1/PLC_1 Instance <-> EtherCAT_1/FG_Transport_EK1100/FG_Transport_Stopper_EL1809_1
//     PlcTask Inputs/MAIN.Machine.FG_Transport.Stopper01.B_Detect.HardwareInput <-> Channel 1/Input
//     PlcTask Inputs/MAIN.Machine.FG_Transport.Stopper02.B_Detect.HardwareInput <-> Channel 5/Input
//     PlcTask Inputs/MAIN.Machine.FG_Transport.Stopper03.B_Detect.HardwareInput <-> Channel 9/Input
//     PlcTask Inputs/MAIN.Machine.FG_Transport.Stopper04.B_Detect.HardwareInput <-> Channel 13/Input
//     PlcTask Inputs/MAIN.Machine.FG_Transport.Stopper01.B_Exit.HardwareInput <-> Channel 2/Input
//     PlcTask Inputs/MAIN.Machine.FG_Transport.Stopper02.B_Exit.HardwareInput <-> Channel 6/Input
//     PlcTask Inputs/MAIN.Machine.FG_Transport.Stopper03.B_Exit.HardwareInput <-> Channel 10/Input
//     PlcTask Inputs/MAIN.Machine.FG_Transport.Stopper04.B_Exit.HardwareInput <-> Channel 14/Input
//     PlcTask Inputs/MAIN.Machine.FG_Transport.Stopper01.Y_Stopper.ExtendedSensor <-> Channel 4/Input
//     PlcTask Inputs/MAIN.Machine.FG_Transport.Stopper02.Y_Stopper.ExtendedSensor <-> Channel 8/Input
//     PlcTask Inputs/MAIN.Machine.FG_Transport.Stopper03.Y_Stopper.ExtendedSensor <-> Channel 12/Input
//     PlcTask Inputs/MAIN.Machine.FG_Transport.Stopper04.Y_Stopper.ExtendedSensor <-> Channel 16/Input
//     PlcTask Inputs/MAIN.Machine.FG_Transport.Stopper01.Y_Stopper.RetractedSensor <-> Channel 3/Input
//     PlcTask Inputs/MAIN.Machine.FG_Transport.Stopper02.Y_Stopper.RetractedSensor <-> Channel 7/Input
//     PlcTask Inputs/MAIN.Machine.FG_Transport.Stopper03.Y_Stopper.RetractedSensor <-> Channel 11/Input
//     PlcTask Inputs/MAIN.Machine.FG_Transport.Stopper04.Y_Stopper.RetractedSensor <-> Channel 15/Input
//   PLC_1/PLC_1 Instance <-> EtherCAT_1/FG_Transport_EK1100/FG_Transport_Stopper_EL2008_1
//     PlcTask Outputs/MAIN.Machine.FG_Transport.Stopper01.Y_Stopper._ExtendOutput <-> Channel 1/Output
//     PlcTask Outputs/MAIN.Machine.FG_Transport.Stopper02.Y_Stopper._ExtendOutput <-> Channel 2/Output
//     PlcTask Outputs/MAIN.Machine.FG_Transport.Stopper03.Y_Stopper._ExtendOutput <-> Channel 3/Output
//     PlcTask Outputs/MAIN.Machine.FG_Transport.Stopper04.Y_Stopper._ExtendOutput <-> Channel 4/Output
//   SIM_1/SIM_1 Instance <-> EtherCAT_1_SIM/FG_01_EL1008_1
//     PlcTask Outputs/GVL_EtherCAT_1_SIM.FG_01_EL1008_1.bIn1 <-> Channel 1/Input
//     PlcTask Outputs/GVL_EtherCAT_1_SIM.FG_01_EL1008_1.bIn2 <-> Channel 2/Input
//     PlcTask Outputs/GVL_EtherCAT_1_SIM.FG_01_EL1008_1.bIn3 <-> Channel 3/Input
//     PlcTask Outputs/GVL_EtherCAT_1_SIM.FG_01_EL1008_1.bIn4 <-> Channel 4/Input
//     PlcTask Outputs/GVL_EtherCAT_1_SIM.FG_01_EL1008_1.bIn5 <-> Channel 5/Input
//     PlcTask Outputs/GVL_EtherCAT_1_SIM.FG_01_EL1008_1.bIn6 <-> Channel 6/Input
//     PlcTask Outputs/GVL_EtherCAT_1_SIM.FG_01_EL1008_1.bIn7 <-> Channel 7/Input
//     PlcTask Outputs/GVL_EtherCAT_1_SIM.FG_01_EL1008_1.bIn8 <-> Channel 8/Input
//   SIM_1/SIM_1 Instance <-> EtherCAT_1_SIM/FG_01_EL1008_2
//     PlcTask Outputs/GVL_EtherCAT_1_SIM.FG_01_EL1008_2.bIn1 <-> Channel 1/Input
//     PlcTask Outputs/GVL_EtherCAT_1_SIM.FG_01_EL1008_2.bIn2 <-> Channel 2/Input
//     PlcTask Outputs/GVL_EtherCAT_1_SIM.FG_01_EL1008_2.bIn3 <-> Channel 3/Input
//     PlcTask Outputs/GVL_EtherCAT_1_SIM.FG_01_EL1008_2.bIn4 <-> Channel 4/Input
//     PlcTask Outputs/GVL_EtherCAT_1_SIM.FG_01_EL1008_2.bIn5 <-> Channel 5/Input
//     PlcTask Outputs/GVL_EtherCAT_1_SIM.FG_01_EL1008_2.bIn6 <-> Channel 6/Input
//     PlcTask Outputs/GVL_EtherCAT_1_SIM.FG_01_EL1008_2.bIn7 <-> Channel 7/Input
//     PlcTask Outputs/GVL_EtherCAT_1_SIM.FG_01_EL1008_2.bIn8 <-> Channel 8/Input
//   SIM_1/SIM_1 Instance <-> EtherCAT_1_SIM/FG_01_EL1859_1
//     PlcTask Inputs/GVL_EtherCAT_1_SIM.FG_01_EL1859_1.bOut1 <-> Channel 9/Output
//     PlcTask Inputs/GVL_EtherCAT_1_SIM.FG_01_EL1859_1.bOut2 <-> Channel 10/Output
//     PlcTask Inputs/GVL_EtherCAT_1_SIM.FG_01_EL1859_1.bOut3 <-> Channel 11/Output
//     PlcTask Inputs/GVL_EtherCAT_1_SIM.FG_01_EL1859_1.bOut4 <-> Channel 12/Output
//     PlcTask Inputs/GVL_EtherCAT_1_SIM.FG_01_EL1859_1.bOut5 <-> Channel 13/Output
//     PlcTask Inputs/GVL_EtherCAT_1_SIM.FG_01_EL1859_1.bOut6 <-> Channel 14/Output
//     PlcTask Inputs/GVL_EtherCAT_1_SIM.FG_01_EL1859_1.bOut7 <-> Channel 15/Output
//     PlcTask Inputs/GVL_EtherCAT_1_SIM.FG_01_EL1859_1.bOut8 <-> Channel 16/Output
//     PlcTask Outputs/GVL_EtherCAT_1_SIM.FG_01_EL1859_1.bIn1 <-> Channel 1/Input
//     PlcTask Outputs/GVL_EtherCAT_1_SIM.FG_01_EL1859_1.bIn2 <-> Channel 2/Input
//     PlcTask Outputs/GVL_EtherCAT_1_SIM.FG_01_EL1859_1.bIn3 <-> Channel 3/Input
//     PlcTask Outputs/GVL_EtherCAT_1_SIM.FG_01_EL1859_1.bIn4 <-> Channel 4/Input
//     PlcTask Outputs/GVL_EtherCAT_1_SIM.FG_01_EL1859_1.bIn5 <-> Channel 5/Input
//     PlcTask Outputs/GVL_EtherCAT_1_SIM.FG_01_EL1859_1.bIn6 <-> Channel 6/Input
//     PlcTask Outputs/GVL_EtherCAT_1_SIM.FG_01_EL1859_1.bIn7 <-> Channel 7/Input
//     PlcTask Outputs/GVL_EtherCAT_1_SIM.FG_01_EL1859_1.bIn8 <-> Channel 8/Input
//   SIM_1/SIM_1 Instance <-> EtherCAT_1_SIM/FG_01_EL1859_2
//     PlcTask Inputs/GVL_EtherCAT_1_SIM.FG_01_EL1859_2.bOut1 <-> Channel 9/Output
//     PlcTask Inputs/GVL_EtherCAT_1_SIM.FG_01_EL1859_2.bOut2 <-> Channel 10/Output
//     PlcTask Inputs/GVL_EtherCAT_1_SIM.FG_01_EL1859_2.bOut3 <-> Channel 11/Output
//     PlcTask Inputs/GVL_EtherCAT_1_SIM.FG_01_EL1859_2.bOut4 <-> Channel 12/Output
//     PlcTask Inputs/GVL_EtherCAT_1_SIM.FG_01_EL1859_2.bOut5 <-> Channel 13/Output
//     PlcTask Inputs/GVL_EtherCAT_1_SIM.FG_01_EL1859_2.bOut6 <-> Channel 14/Output
//     PlcTask Inputs/GVL_EtherCAT_1_SIM.FG_01_EL1859_2.bOut7 <-> Channel 15/Output
//     PlcTask Inputs/GVL_EtherCAT_1_SIM.FG_01_EL1859_2.bOut8 <-> Channel 16/Output
//     PlcTask Outputs/GVL_EtherCAT_1_SIM.FG_01_EL1859_2.bIn1 <-> Channel 1/Input
//     PlcTask Outputs/GVL_EtherCAT_1_SIM.FG_01_EL1859_2.bIn2 <-> Channel 2/Input
//     PlcTask Outputs/GVL_EtherCAT_1_SIM.FG_01_EL1859_2.bIn3 <-> Channel 3/Input
//     PlcTask Outputs/GVL_EtherCAT_1_SIM.FG_01_EL1859_2.bIn4 <-> Channel 4/Input
//     PlcTask Outputs/GVL_EtherCAT_1_SIM.FG_01_EL1859_2.bIn5 <-> Channel 5/Input
//     PlcTask Outputs/GVL_EtherCAT_1_SIM.FG_01_EL1859_2.bIn6 <-> Channel 6/Input
//     PlcTask Outputs/GVL_EtherCAT_1_SIM.FG_01_EL1859_2.bIn7 <-> Channel 7/Input
//     PlcTask Outputs/GVL_EtherCAT_1_SIM.FG_01_EL1859_2.bIn8 <-> Channel 8/Input
//   SIM_1/SIM_1 Instance <-> EtherCAT_1_SIM/FG_01_EL2008_1
//     PlcTask Inputs/GVL_EtherCAT_1_SIM.FG_01_EL2008_1.bOut1 <-> Channel 1/Output
//     PlcTask Inputs/GVL_EtherCAT_1_SIM.FG_01_EL2008_1.bOut2 <-> Channel 2/Output
//     PlcTask Inputs/GVL_EtherCAT_1_SIM.FG_01_EL2008_1.bOut3 <-> Channel 3/Output
//     PlcTask Inputs/GVL_EtherCAT_1_SIM.FG_01_EL2008_1.bOut4 <-> Channel 4/Output
//     PlcTask Inputs/GVL_EtherCAT_1_SIM.FG_01_EL2008_1.bOut5 <-> Channel 5/Output
//     PlcTask Inputs/GVL_EtherCAT_1_SIM.FG_01_EL2008_1.bOut6 <-> Channel 6/Output
//     PlcTask Inputs/GVL_EtherCAT_1_SIM.FG_01_EL2008_1.bOut7 <-> Channel 7/Output
//     PlcTask Inputs/GVL_EtherCAT_1_SIM.FG_01_EL2008_1.bOut8 <-> Channel 8/Output
//   SIM_1/SIM_1 Instance <-> EtherCAT_1_SIM/FG_02_EL1859_1
//     PlcTask Inputs/GVL_EtherCAT_1_SIM.FG_02_EL1859_1.bOut1 <-> Channel 9/Output
//     PlcTask Inputs/GVL_EtherCAT_1_SIM.FG_02_EL1859_1.bOut2 <-> Channel 10/Output
//     PlcTask Inputs/GVL_EtherCAT_1_SIM.FG_02_EL1859_1.bOut3 <-> Channel 11/Output
//     PlcTask Inputs/GVL_EtherCAT_1_SIM.FG_02_EL1859_1.bOut4 <-> Channel 12/Output
//     PlcTask Inputs/GVL_EtherCAT_1_SIM.FG_02_EL1859_1.bOut5 <-> Channel 13/Output
//     PlcTask Inputs/GVL_EtherCAT_1_SIM.FG_02_EL1859_1.bOut6 <-> Channel 14/Output
//     PlcTask Inputs/GVL_EtherCAT_1_SIM.FG_02_EL1859_1.bOut7 <-> Channel 15/Output
//     PlcTask Inputs/GVL_EtherCAT_1_SIM.FG_02_EL1859_1.bOut8 <-> Channel 16/Output
//     PlcTask Outputs/GVL_EtherCAT_1_SIM.FG_02_EL1859_1.bIn1 <-> Channel 1/Input
//     PlcTask Outputs/GVL_EtherCAT_1_SIM.FG_02_EL1859_1.bIn2 <-> Channel 2/Input
//     PlcTask Outputs/GVL_EtherCAT_1_SIM.FG_02_EL1859_1.bIn3 <-> Channel 3/Input
//     PlcTask Outputs/GVL_EtherCAT_1_SIM.FG_02_EL1859_1.bIn4 <-> Channel 4/Input
//     PlcTask Outputs/GVL_EtherCAT_1_SIM.FG_02_EL1859_1.bIn5 <-> Channel 5/Input
//     PlcTask Outputs/GVL_EtherCAT_1_SIM.FG_02_EL1859_1.bIn6 <-> Channel 6/Input
//     PlcTask Outputs/GVL_EtherCAT_1_SIM.FG_02_EL1859_1.bIn7 <-> Channel 7/Input
//     PlcTask Outputs/GVL_EtherCAT_1_SIM.FG_02_EL1859_1.bIn8 <-> Channel 8/Input
//   SIM_1/SIM_1 Instance <-> EtherCAT_1_SIM/FG_03_EL1809_1
//     PlcTask Outputs/GVL_EtherCAT_1_SIM.FG_03_EL1809_1.bIn1 <-> Channel 1/Input
//     PlcTask Outputs/GVL_EtherCAT_1_SIM.FG_03_EL1809_1.bIn10 <-> Channel 10/Input
//     PlcTask Outputs/GVL_EtherCAT_1_SIM.FG_03_EL1809_1.bIn11 <-> Channel 11/Input
//     PlcTask Outputs/GVL_EtherCAT_1_SIM.FG_03_EL1809_1.bIn12 <-> Channel 12/Input
//     PlcTask Outputs/GVL_EtherCAT_1_SIM.FG_03_EL1809_1.bIn13 <-> Channel 13/Input
//     PlcTask Outputs/GVL_EtherCAT_1_SIM.FG_03_EL1809_1.bIn14 <-> Channel 14/Input
//     PlcTask Outputs/GVL_EtherCAT_1_SIM.FG_03_EL1809_1.bIn15 <-> Channel 15/Input
//     PlcTask Outputs/GVL_EtherCAT_1_SIM.FG_03_EL1809_1.bIn16 <-> Channel 16/Input
//     PlcTask Outputs/GVL_EtherCAT_1_SIM.FG_03_EL1809_1.bIn2 <-> Channel 2/Input
//     PlcTask Outputs/GVL_EtherCAT_1_SIM.FG_03_EL1809_1.bIn3 <-> Channel 3/Input
//     PlcTask Outputs/GVL_EtherCAT_1_SIM.FG_03_EL1809_1.bIn4 <-> Channel 4/Input
//     PlcTask Outputs/GVL_EtherCAT_1_SIM.FG_03_EL1809_1.bIn5 <-> Channel 5/Input
//     PlcTask Outputs/GVL_EtherCAT_1_SIM.FG_03_EL1809_1.bIn6 <-> Channel 6/Input
//     PlcTask Outputs/GVL_EtherCAT_1_SIM.FG_03_EL1809_1.bIn7 <-> Channel 7/Input
//     PlcTask Outputs/GVL_EtherCAT_1_SIM.FG_03_EL1809_1.bIn8 <-> Channel 8/Input
//     PlcTask Outputs/GVL_EtherCAT_1_SIM.FG_03_EL1809_1.bIn9 <-> Channel 9/Input
//   SIM_1/SIM_1 Instance <-> EtherCAT_1_SIM/FG_03_EL2809_1
//     PlcTask Inputs/GVL_EtherCAT_1_SIM.FG_03_EL2809_1.bOut1 <-> Channel 1/Output
//     PlcTask Inputs/GVL_EtherCAT_1_SIM.FG_03_EL2809_1.bOut10 <-> Channel 10/Output
//     PlcTask Inputs/GVL_EtherCAT_1_SIM.FG_03_EL2809_1.bOut11 <-> Channel 11/Output
//     PlcTask Inputs/GVL_EtherCAT_1_SIM.FG_03_EL2809_1.bOut12 <-> Channel 12/Output
//     PlcTask Inputs/GVL_EtherCAT_1_SIM.FG_03_EL2809_1.bOut13 <-> Channel 13/Output
//     PlcTask Inputs/GVL_EtherCAT_1_SIM.FG_03_EL2809_1.bOut14 <-> Channel 14/Output
//     PlcTask Inputs/GVL_EtherCAT_1_SIM.FG_03_EL2809_1.bOut15 <-> Channel 15/Output
//     PlcTask Inputs/GVL_EtherCAT_1_SIM.FG_03_EL2809_1.bOut16 <-> Channel 16/Output
//     PlcTask Inputs/GVL_EtherCAT_1_SIM.FG_03_EL2809_1.bOut2 <-> Channel 2/Output
//     PlcTask Inputs/GVL_EtherCAT_1_SIM.FG_03_EL2809_1.bOut3 <-> Channel 3/Output
//     PlcTask Inputs/GVL_EtherCAT_1_SIM.FG_03_EL2809_1.bOut4 <-> Channel 4/Output
//     PlcTask Inputs/GVL_EtherCAT_1_SIM.FG_03_EL2809_1.bOut5 <-> Channel 5/Output
//     PlcTask Inputs/GVL_EtherCAT_1_SIM.FG_03_EL2809_1.bOut6 <-> Channel 6/Output
//     PlcTask Inputs/GVL_EtherCAT_1_SIM.FG_03_EL2809_1.bOut7 <-> Channel 7/Output
//     PlcTask Inputs/GVL_EtherCAT_1_SIM.FG_03_EL2809_1.bOut8 <-> Channel 8/Output
//     PlcTask Inputs/GVL_EtherCAT_1_SIM.FG_03_EL2809_1.bOut9 <-> Channel 9/Output
//   SIM_1/SIM_1 Instance <-> EtherCAT_1_SIM/FG_04_EL1008_1
//     PlcTask Outputs/GVL_EtherCAT_1_SIM.FG_04_EL1008_1.bIn1 <-> Channel 1/Input
//     PlcTask Outputs/GVL_EtherCAT_1_SIM.FG_04_EL1008_1.bIn2 <-> Channel 2/Input
//     PlcTask Outputs/GVL_EtherCAT_1_SIM.FG_04_EL1008_1.bIn3 <-> Channel 3/Input
//     PlcTask Outputs/GVL_EtherCAT_1_SIM.FG_04_EL1008_1.bIn4 <-> Channel 4/Input
//     PlcTask Outputs/GVL_EtherCAT_1_SIM.FG_04_EL1008_1.bIn5 <-> Channel 5/Input
//     PlcTask Outputs/GVL_EtherCAT_1_SIM.FG_04_EL1008_1.bIn6 <-> Channel 6/Input
//     PlcTask Outputs/GVL_EtherCAT_1_SIM.FG_04_EL1008_1.bIn7 <-> Channel 7/Input
//     PlcTask Outputs/GVL_EtherCAT_1_SIM.FG_04_EL1008_1.bIn8 <-> Channel 8/Input
//   SIM_1/SIM_1 Instance <-> EtherCAT_1_SIM/FG_04_EL2008_1
//     PlcTask Inputs/GVL_EtherCAT_1_SIM.FG_04_EL2008_1.bOut1 <-> Channel 1/Output
//     PlcTask Inputs/GVL_EtherCAT_1_SIM.FG_04_EL2008_1.bOut2 <-> Channel 2/Output
//     PlcTask Inputs/GVL_EtherCAT_1_SIM.FG_04_EL2008_1.bOut3 <-> Channel 3/Output
//     PlcTask Inputs/GVL_EtherCAT_1_SIM.FG_04_EL2008_1.bOut4 <-> Channel 4/Output
//     PlcTask Inputs/GVL_EtherCAT_1_SIM.FG_04_EL2008_1.bOut5 <-> Channel 5/Output
//     PlcTask Inputs/GVL_EtherCAT_1_SIM.FG_04_EL2008_1.bOut6 <-> Channel 6/Output
//     PlcTask Inputs/GVL_EtherCAT_1_SIM.FG_04_EL2008_1.bOut7 <-> Channel 7/Output
//     PlcTask Inputs/GVL_EtherCAT_1_SIM.FG_04_EL2008_1.bOut8 <-> Channel 8/Output
//   SIM_1/SIM_1 Instance <-> EtherCAT_1_SIM/FG_05_EL1809_1
//     PlcTask Outputs/GVL_EtherCAT_1_SIM.FG_05_EL1809_1.bIn1 <-> Channel 1/Input
//     PlcTask Outputs/GVL_EtherCAT_1_SIM.FG_05_EL1809_1.bIn10 <-> Channel 10/Input
//     PlcTask Outputs/GVL_EtherCAT_1_SIM.FG_05_EL1809_1.bIn11 <-> Channel 11/Input
//     PlcTask Outputs/GVL_EtherCAT_1_SIM.FG_05_EL1809_1.bIn12 <-> Channel 12/Input
//     PlcTask Outputs/GVL_EtherCAT_1_SIM.FG_05_EL1809_1.bIn13 <-> Channel 13/Input
//     PlcTask Outputs/GVL_EtherCAT_1_SIM.FG_05_EL1809_1.bIn14 <-> Channel 14/Input
//     PlcTask Outputs/GVL_EtherCAT_1_SIM.FG_05_EL1809_1.bIn15 <-> Channel 15/Input
//     PlcTask Outputs/GVL_EtherCAT_1_SIM.FG_05_EL1809_1.bIn16 <-> Channel 16/Input
//     PlcTask Outputs/GVL_EtherCAT_1_SIM.FG_05_EL1809_1.bIn2 <-> Channel 2/Input
//     PlcTask Outputs/GVL_EtherCAT_1_SIM.FG_05_EL1809_1.bIn3 <-> Channel 3/Input
//     PlcTask Outputs/GVL_EtherCAT_1_SIM.FG_05_EL1809_1.bIn4 <-> Channel 4/Input
//     PlcTask Outputs/GVL_EtherCAT_1_SIM.FG_05_EL1809_1.bIn5 <-> Channel 5/Input
//     PlcTask Outputs/GVL_EtherCAT_1_SIM.FG_05_EL1809_1.bIn6 <-> Channel 6/Input
//     PlcTask Outputs/GVL_EtherCAT_1_SIM.FG_05_EL1809_1.bIn7 <-> Channel 7/Input
//     PlcTask Outputs/GVL_EtherCAT_1_SIM.FG_05_EL1809_1.bIn8 <-> Channel 8/Input
//     PlcTask Outputs/GVL_EtherCAT_1_SIM.FG_05_EL1809_1.bIn9 <-> Channel 9/Input
//   SIM_1/SIM_1 Instance <-> EtherCAT_1_SIM/FG_05_EL1859_1
//     PlcTask Inputs/GVL_EtherCAT_1_SIM.FG_05_EL1859_1.bOut1 <-> Channel 9/Output
//     PlcTask Inputs/GVL_EtherCAT_1_SIM.FG_05_EL1859_1.bOut2 <-> Channel 10/Output
//     PlcTask Inputs/GVL_EtherCAT_1_SIM.FG_05_EL1859_1.bOut3 <-> Channel 11/Output
//     PlcTask Inputs/GVL_EtherCAT_1_SIM.FG_05_EL1859_1.bOut4 <-> Channel 12/Output
//     PlcTask Inputs/GVL_EtherCAT_1_SIM.FG_05_EL1859_1.bOut5 <-> Channel 13/Output
//     PlcTask Inputs/GVL_EtherCAT_1_SIM.FG_05_EL1859_1.bOut6 <-> Channel 14/Output
//     PlcTask Inputs/GVL_EtherCAT_1_SIM.FG_05_EL1859_1.bOut7 <-> Channel 15/Output
//     PlcTask Inputs/GVL_EtherCAT_1_SIM.FG_05_EL1859_1.bOut8 <-> Channel 16/Output
//     PlcTask Outputs/GVL_EtherCAT_1_SIM.FG_05_EL1859_1.bIn1 <-> Channel 1/Input
//     PlcTask Outputs/GVL_EtherCAT_1_SIM.FG_05_EL1859_1.bIn2 <-> Channel 2/Input
//     PlcTask Outputs/GVL_EtherCAT_1_SIM.FG_05_EL1859_1.bIn3 <-> Channel 3/Input
//     PlcTask Outputs/GVL_EtherCAT_1_SIM.FG_05_EL1859_1.bIn4 <-> Channel 4/Input
//     PlcTask Outputs/GVL_EtherCAT_1_SIM.FG_05_EL1859_1.bIn5 <-> Channel 5/Input
//     PlcTask Outputs/GVL_EtherCAT_1_SIM.FG_05_EL1859_1.bIn6 <-> Channel 6/Input
//     PlcTask Outputs/GVL_EtherCAT_1_SIM.FG_05_EL1859_1.bIn7 <-> Channel 7/Input
//     PlcTask Outputs/GVL_EtherCAT_1_SIM.FG_05_EL1859_1.bIn8 <-> Channel 8/Input
//   SIM_1/SIM_1 Instance <-> EtherCAT_1_SIM/FG_05_EL1859_2
//     PlcTask Inputs/GVL_EtherCAT_1_SIM.FG_05_EL1859_2.bOut1 <-> Channel 9/Output
//     PlcTask Inputs/GVL_EtherCAT_1_SIM.FG_05_EL1859_2.bOut2 <-> Channel 10/Output
//     PlcTask Inputs/GVL_EtherCAT_1_SIM.FG_05_EL1859_2.bOut3 <-> Channel 11/Output
//     PlcTask Inputs/GVL_EtherCAT_1_SIM.FG_05_EL1859_2.bOut4 <-> Channel 12/Output
//     PlcTask Inputs/GVL_EtherCAT_1_SIM.FG_05_EL1859_2.bOut5 <-> Channel 13/Output
//     PlcTask Inputs/GVL_EtherCAT_1_SIM.FG_05_EL1859_2.bOut6 <-> Channel 14/Output
//     PlcTask Inputs/GVL_EtherCAT_1_SIM.FG_05_EL1859_2.bOut7 <-> Channel 15/Output
//     PlcTask Inputs/GVL_EtherCAT_1_SIM.FG_05_EL1859_2.bOut8 <-> Channel 16/Output
//     PlcTask Outputs/GVL_EtherCAT_1_SIM.FG_05_EL1859_2.bIn1 <-> Channel 1/Input
//     PlcTask Outputs/GVL_EtherCAT_1_SIM.FG_05_EL1859_2.bIn2 <-> Channel 2/Input
//     PlcTask Outputs/GVL_EtherCAT_1_SIM.FG_05_EL1859_2.bIn3 <-> Channel 3/Input
//     PlcTask Outputs/GVL_EtherCAT_1_SIM.FG_05_EL1859_2.bIn4 <-> Channel 4/Input
//     PlcTask Outputs/GVL_EtherCAT_1_SIM.FG_05_EL1859_2.bIn5 <-> Channel 5/Input
//     PlcTask Outputs/GVL_EtherCAT_1_SIM.FG_05_EL1859_2.bIn6 <-> Channel 6/Input
//     PlcTask Outputs/GVL_EtherCAT_1_SIM.FG_05_EL1859_2.bIn7 <-> Channel 7/Input
//     PlcTask Outputs/GVL_EtherCAT_1_SIM.FG_05_EL1859_2.bIn8 <-> Channel 8/Input
//   SIM_1/SIM_1 Instance <-> EtherCAT_1_SIM/FG_05_EL2809_1
//     PlcTask Inputs/GVL_EtherCAT_1_SIM.FG_05_EL2809_1.bOut1 <-> Channel 1/Output
//     PlcTask Inputs/GVL_EtherCAT_1_SIM.FG_05_EL2809_1.bOut10 <-> Channel 10/Output
//     PlcTask Inputs/GVL_EtherCAT_1_SIM.FG_05_EL2809_1.bOut11 <-> Channel 11/Output
//     PlcTask Inputs/GVL_EtherCAT_1_SIM.FG_05_EL2809_1.bOut12 <-> Channel 12/Output
//     PlcTask Inputs/GVL_EtherCAT_1_SIM.FG_05_EL2809_1.bOut13 <-> Channel 13/Output
//     PlcTask Inputs/GVL_EtherCAT_1_SIM.FG_05_EL2809_1.bOut14 <-> Channel 14/Output
//     PlcTask Inputs/GVL_EtherCAT_1_SIM.FG_05_EL2809_1.bOut15 <-> Channel 15/Output
//     PlcTask Inputs/GVL_EtherCAT_1_SIM.FG_05_EL2809_1.bOut16 <-> Channel 16/Output
//     PlcTask Inputs/GVL_EtherCAT_1_SIM.FG_05_EL2809_1.bOut2 <-> Channel 2/Output
//     PlcTask Inputs/GVL_EtherCAT_1_SIM.FG_05_EL2809_1.bOut3 <-> Channel 3/Output
//     PlcTask Inputs/GVL_EtherCAT_1_SIM.FG_05_EL2809_1.bOut4 <-> Channel 4/Output
//     PlcTask Inputs/GVL_EtherCAT_1_SIM.FG_05_EL2809_1.bOut5 <-> Channel 5/Output
//     PlcTask Inputs/GVL_EtherCAT_1_SIM.FG_05_EL2809_1.bOut6 <-> Channel 6/Output
//     PlcTask Inputs/GVL_EtherCAT_1_SIM.FG_05_EL2809_1.bOut7 <-> Channel 7/Output
//     PlcTask Inputs/GVL_EtherCAT_1_SIM.FG_05_EL2809_1.bOut8 <-> Channel 8/Output
//     PlcTask Inputs/GVL_EtherCAT_1_SIM.FG_05_EL2809_1.bOut9 <-> Channel 9/Output
//   SIM_1/SIM_1 Instance <-> EtherCAT_1_SIM/FG_System_Door_EL1809_1
//     PlcTask Outputs/GVL_EtherCAT_1_SIM.FG_System_Door_EL1809_1.bIn{1..16} <-> Channel {1..16}/Input  (16 links)
//   SIM_1/SIM_1 Instance <-> EtherCAT_1_SIM/FG_System_Door_EL2008_1
//     PlcTask Inputs/GVL_EtherCAT_1_SIM.FG_System_Door_EL2008_1.bOut{1..8} <-> Channel {1..8}/Output  (8 links)
//   SIM_1/SIM_1 Instance <-> EtherCAT_1_SIM/FG_System_Panel_EL1809_1
//     PlcTask Outputs/GVL_EtherCAT_1_SIM.FG_System_Panel_EL1809_1.bIn{1..16} <-> Channel {1..16}/Input  (16 links)
//   SIM_1/SIM_1 Instance <-> EtherCAT_1_SIM/FG_System_Panel_EL2809_1
//     PlcTask Inputs/GVL_EtherCAT_1_SIM.FG_System_Panel_EL2809_1.bOut{1..16} <-> Channel {1..16}/Output  (16 links)
//   SIM_1/SIM_1 Instance <-> EtherCAT_1_SIM/FG_Transport_Drive_EL1008_1
//     PlcTask Outputs/GVL_EtherCAT_1_SIM.FG_Transport_Drive_EL1008_1.bIn{1..8} <-> Channel {1..8}/Input  (8 links)
//   SIM_1/SIM_1 Instance <-> EtherCAT_1_SIM/FG_Transport_Drive_EL2008_1
//     PlcTask Inputs/GVL_EtherCAT_1_SIM.FG_Transport_Drive_EL2008_1.bOut{1..8} <-> Channel {1..8}/Output  (8 links)
//   SIM_1/SIM_1 Instance <-> EtherCAT_1_SIM/FG_Transport_Index_EL1809_1
//     PlcTask Outputs/GVL_EtherCAT_1_SIM.FG_Transport_Index_EL1809_1.bIn{1..16} <-> Channel {1..16}/Input  (16 links)
//   SIM_1/SIM_1 Instance <-> EtherCAT_1_SIM/FG_Transport_Index_EL1809_2
//     PlcTask Outputs/GVL_EtherCAT_1_SIM.FG_Transport_Index_EL1809_2.bIn{1..16} <-> Channel {1..16}/Input  (16 links)
//   SIM_1/SIM_1 Instance <-> EtherCAT_1_SIM/FG_Transport_Index_EL2809_1
//     PlcTask Inputs/GVL_EtherCAT_1_SIM.FG_Transport_Index_EL2809_1.bOut{1..16} <-> Channel {1..16}/Output  (16 links)
//   SIM_1/SIM_1 Instance <-> EtherCAT_1_SIM/FG_Transport_Lift_EL1809_1
//     PlcTask Outputs/GVL_EtherCAT_1_SIM.FG_Transport_Lift_EL1809_1.bIn{1..16} <-> Channel {1..16}/Input  (16 links)
//   SIM_1/SIM_1 Instance <-> EtherCAT_1_SIM/FG_Transport_Lift_EL2008_1
//     PlcTask Inputs/GVL_EtherCAT_1_SIM.FG_Transport_Lift_EL2008_1.bOut{1..8} <-> Channel {1..8}/Output  (8 links)
//   SIM_1/SIM_1 Instance <-> EtherCAT_1_SIM/FG_Transport_Stopper_EL1809_1
//     PlcTask Outputs/GVL_EtherCAT_1_SIM.FG_Transport_Stopper_EL1809_1.bIn{1..16} <-> Channel {1..16}/Input  (16 links)
//   SIM_1/SIM_1 Instance <-> EtherCAT_1_SIM/FG_Transport_Stopper_EL2008_1
//     PlcTask Inputs/GVL_EtherCAT_1_SIM.FG_Transport_Stopper_EL2008_1.bOut{1..8} <-> Channel {1..8}/Output  (8 links)

// ---- Hil/EtherCAT_1_SIM/GVL_EtherCAT_1_SIM.TcGVL
{attribute 'linkalways'}
{attribute 'qualified_only'}
{attribute 'subsequent'}
{attribute 'pack_mode' := '1'}
VAR_GLOBAL
{attribute 'TcLinkTo' := '
.bIn1 := TIIB(45)^Channel 1^Input;
.bIn2 := TIIB(45)^Channel 2^Input;
.bIn3 := TIIB(45)^Channel 3^Input;
.bIn4 := TIIB(45)^Channel 4^Input;
.bIn5 := TIIB(45)^Channel 5^Input;
.bIn6 := TIIB(45)^Channel 6^Input;
.bIn7 := TIIB(45)^Channel 7^Input;
.bIn8 := TIIB(45)^Channel 8^Input;
.bIn9 := TIIB(45)^Channel 9^Input;
.bIn10 := TIIB(45)^Channel 10^Input;
.bIn11 := TIIB(45)^Channel 11^Input;
.bIn12 := TIIB(45)^Channel 12^Input;
.bIn13 := TIIB(45)^Channel 13^Input;
.bIn14 := TIIB(45)^Channel 14^Input;
.bIn15 := TIIB(45)^Channel 15^Input;
.bIn16 := TIIB(45)^Channel 16^Input'}
FG_System_Panel_EL1809_1 : ST_Beckhoff_16DI;
{attribute 'TcLinkTo' := '
.bOut1 := TIIB(46)^Channel 1^Output;
.bOut2 := TIIB(46)^Channel 2^Output;
.bOut3 := TIIB(46)^Channel 3^Output;
.bOut4 := TIIB(46)^Channel 4^Output;
.bOut5 := TIIB(46)^Channel 5^Output;
.bOut6 := TIIB(46)^Channel 6^Output;
.bOut7 := TIIB(46)^Channel 7^Output;
.bOut8 := TIIB(46)^Channel 8^Output;
.bOut9 := TIIB(46)^Channel 9^Output;
.bOut10 := TIIB(46)^Channel 10^Output;
.bOut11 := TIIB(46)^Channel 11^Output;
.bOut12 := TIIB(46)^Channel 12^Output;
.bOut13 := TIIB(46)^Channel 13^Output;
.bOut14 := TIIB(46)^Channel 14^Output;
.bOut15 := TIIB(46)^Channel 15^Output;
.bOut16 := TIIB(46)^Channel 16^Output'}
FG_System_Panel_EL2809_1 : ST_Beckhoff_16DO;
{attribute 'TcLinkTo' := '
.bIn1 := TIIB(59)^Channel 1^Input;
.bIn2 := TIIB(59)^Channel 2^Input;
.bIn3 := TIIB(59)^Channel 3^Input;
.bIn4 := TIIB(59)^Channel 4^Input;
.bIn5 := TIIB(59)^Channel 5^Input;
.bIn6 := TIIB(59)^Channel 6^Input;
.bIn7 := TIIB(59)^Channel 7^Input;
.bIn8 := TIIB(59)^Channel 8^Input;
.bIn9 := TIIB(59)^Channel 9^Input;
.bIn10 := TIIB(59)^Channel 10^Input;
.bIn11 := TIIB(59)^Channel 11^Input;
.bIn12 := TIIB(59)^Channel 12^Input;
.bIn13 := TIIB(59)^Channel 13^Input;
.bIn14 := TIIB(59)^Channel 14^Input;
.bIn15 := TIIB(59)^Channel 15^Input;
.bIn16 := TIIB(59)^Channel 16^Input'}
FG_System_Door_EL1809_1 : ST_Beckhoff_16DI;
{attribute 'TcLinkTo' := '
.bOut1 := TIIB(60)^Channel 1^Output;
.bOut2 := TIIB(60)^Channel 2^Output;
.bOut3 := TIIB(60)^Channel 3^Output;
.bOut4 := TIIB(60)^Channel 4^Output;
.bOut5 := TIIB(60)^Channel 5^Output;
.bOut6 := TIIB(60)^Channel 6^Output;
.bOut7 := TIIB(60)^Channel 7^Output;
.bOut8 := TIIB(60)^Channel 8^Output'}
FG_System_Door_EL2008_1 : ST_Beckhoff_8DO;
{attribute 'TcLinkTo' := '
.bIn1 := TIIB(62)^Channel 1^Input;
.bIn2 := TIIB(62)^Channel 2^Input;
.bIn3 := TIIB(62)^Channel 3^Input;
.bIn4 := TIIB(62)^Channel 4^Input;
.bIn5 := TIIB(62)^Channel 5^Input;
.bIn6 := TIIB(62)^Channel 6^Input;
.bIn7 := TIIB(62)^Channel 7^Input;
.bIn8 := TIIB(62)^Channel 8^Input;
.bIn9 := TIIB(62)^Channel 9^Input;
.bIn10 := TIIB(62)^Channel 10^Input;
.bIn11 := TIIB(62)^Channel 11^Input;
.bIn12 := TIIB(62)^Channel 12^Input;
.bIn13 := TIIB(62)^Channel 13^Input;
.bIn14 := TIIB(62)^Channel 14^Input;
.bIn15 := TIIB(62)^Channel 15^Input;
.bIn16 := TIIB(62)^Channel 16^Input'}
FG_Transport_Index_EL1809_1 : ST_Beckhoff_16DI;
{attribute 'TcLinkTo' := '
.bIn1 := TIIB(63)^Channel 1^Input;
.bIn2 := TIIB(63)^Channel 2^Input;
.bIn3 := TIIB(63)^Channel 3^Input;
.bIn4 := TIIB(63)^Channel 4^Input;
.bIn5 := TIIB(63)^Channel 5^Input;
.bIn6 := TIIB(63)^Channel 6^Input;
.bIn7 := TIIB(63)^Channel 7^Input;
.bIn8 := TIIB(63)^Channel 8^Input;
.bIn9 := TIIB(63)^Channel 9^Input;
.bIn10 := TIIB(63)^Channel 10^Input;
.bIn11 := TIIB(63)^Channel 11^Input;
.bIn12 := TIIB(63)^Channel 12^Input;
.bIn13 := TIIB(63)^Channel 13^Input;
.bIn14 := TIIB(63)^Channel 14^Input;
.bIn15 := TIIB(63)^Channel 15^Input;
.bIn16 := TIIB(63)^Channel 16^Input'}
FG_Transport_Index_EL1809_2 : ST_Beckhoff_16DI;
{attribute 'TcLinkTo' := '
.bIn1 := TIIB(64)^Channel 1^Input;
.bIn2 := TIIB(64)^Channel 2^Input;
.bIn3 := TIIB(64)^Channel 3^Input;
.bIn4 := TIIB(64)^Channel 4^Input;
.bIn5 := TIIB(64)^Channel 5^Input;
.bIn6 := TIIB(64)^Channel 6^Input;
.bIn7 := TIIB(64)^Channel 7^Input;
.bIn8 := TIIB(64)^Channel 8^Input;
.bIn9 := TIIB(64)^Channel 9^Input;
.bIn10 := TIIB(64)^Channel 10^Input;
.bIn11 := TIIB(64)^Channel 11^Input;
.bIn12 := TIIB(64)^Channel 12^Input;
.bIn13 := TIIB(64)^Channel 13^Input;
.bIn14 := TIIB(64)^Channel 14^Input;
.bIn15 := TIIB(64)^Channel 15^Input;
.bIn16 := TIIB(64)^Channel 16^Input'}
FG_Transport_Stopper_EL1809_1 : ST_Beckhoff_16DI;
{attribute 'TcLinkTo' := '
.bIn1 := TIIB(65)^Channel 1^Input;
.bIn2 := TIIB(65)^Channel 2^Input;
.bIn3 := TIIB(65)^Channel 3^Input;
.bIn4 := TIIB(65)^Channel 4^Input;
.bIn5 := TIIB(65)^Channel 5^Input;
.bIn6 := TIIB(65)^Channel 6^Input;
.bIn7 := TIIB(65)^Channel 7^Input;
.bIn8 := TIIB(65)^Channel 8^Input;
.bIn9 := TIIB(65)^Channel 9^Input;
.bIn10 := TIIB(65)^Channel 10^Input;
.bIn11 := TIIB(65)^Channel 11^Input;
.bIn12 := TIIB(65)^Channel 12^Input;
.bIn13 := TIIB(65)^Channel 13^Input;
.bIn14 := TIIB(65)^Channel 14^Input;
.bIn15 := TIIB(65)^Channel 15^Input;
.bIn16 := TIIB(65)^Channel 16^Input'}
FG_Transport_Lift_EL1809_1 : ST_Beckhoff_16DI;
{attribute 'TcLinkTo' := '
.bIn1 := TIIB(66)^Channel 1^Input;
.bIn2 := TIIB(66)^Channel 2^Input;
.bIn3 := TIIB(66)^Channel 3^Input;
.bIn4 := TIIB(66)^Channel 4^Input;
.bIn5 := TIIB(66)^Channel 5^Input;
.bIn6 := TIIB(66)^Channel 6^Input;
.bIn7 := TIIB(66)^Channel 7^Input;
.bIn8 := TIIB(66)^Channel 8^Input'}
FG_Transport_Drive_EL1008_1 : ST_Beckhoff_8DI;
{attribute 'TcLinkTo' := '
.bOut1 := TIIB(67)^Channel 1^Output;
.bOut2 := TIIB(67)^Channel 2^Output;
.bOut3 := TIIB(67)^Channel 3^Output;
.bOut4 := TIIB(67)^Channel 4^Output;
.bOut5 := TIIB(67)^Channel 5^Output;
.bOut6 := TIIB(67)^Channel 6^Output;
.bOut7 := TIIB(67)^Channel 7^Output;
.bOut8 := TIIB(67)^Channel 8^Output;
.bOut9 := TIIB(67)^Channel 9^Output;
.bOut10 := TIIB(67)^Channel 10^Output;
.bOut11 := TIIB(67)^Channel 11^Output;
.bOut12 := TIIB(67)^Channel 12^Output;
.bOut13 := TIIB(67)^Channel 13^Output;
.bOut14 := TIIB(67)^Channel 14^Output;
.bOut15 := TIIB(67)^Channel 15^Output;
.bOut16 := TIIB(67)^Channel 16^Output'}
FG_Transport_Index_EL2809_1 : ST_Beckhoff_16DO;
{attribute 'TcLinkTo' := '
.bOut1 := TIIB(68)^Channel 1^Output;
.bOut2 := TIIB(68)^Channel 2^Output;
.bOut3 := TIIB(68)^Channel 3^Output;
.bOut4 := TIIB(68)^Channel 4^Output;
.bOut5 := TIIB(68)^Channel 5^Output;
.bOut6 := TIIB(68)^Channel 6^Output;
.bOut7 := TIIB(68)^Channel 7^Output;
.bOut8 := TIIB(68)^Channel 8^Output'}
FG_Transport_Stopper_EL2008_1 : ST_Beckhoff_8DO;
{attribute 'TcLinkTo' := '
.bOut1 := TIIB(69)^Channel 1^Output;
.bOut2 := TIIB(69)^Channel 2^Output;
.bOut3 := TIIB(69)^Channel 3^Output;
.bOut4 := TIIB(69)^Channel 4^Output;
.bOut5 := TIIB(69)^Channel 5^Output;
.bOut6 := TIIB(69)^Channel 6^Output;
.bOut7 := TIIB(69)^Channel 7^Output;
.bOut8 := TIIB(69)^Channel 8^Output'}
FG_Transport_Lift_EL2008_1 : ST_Beckhoff_8DO;
{attribute 'TcLinkTo' := '
.bOut1 := TIIB(70)^Channel 1^Output;
.bOut2 := TIIB(70)^Channel 2^Output;
.bOut3 := TIIB(70)^Channel 3^Output;
.bOut4 := TIIB(70)^Channel 4^Output;
.bOut5 := TIIB(70)^Channel 5^Output;
.bOut6 := TIIB(70)^Channel 6^Output;
.bOut7 := TIIB(70)^Channel 7^Output;
.bOut8 := TIIB(70)^Channel 8^Output'}
FG_Transport_Drive_EL2008_1 : ST_Beckhoff_8DO;
{attribute 'TcLinkTo' := '
.bIn1 := TIIB(72)^Channel 1^Input;
.bIn2 := TIIB(72)^Channel 2^Input;
.bIn3 := TIIB(72)^Channel 3^Input;
.bIn4 := TIIB(72)^Channel 4^Input;
.bIn5 := TIIB(72)^Channel 5^Input;
.bIn6 := TIIB(72)^Channel 6^Input;
.bIn7 := TIIB(72)^Channel 7^Input;
.bIn8 := TIIB(72)^Channel 8^Input'}
FG_01_EL1008_1 : ST_Beckhoff_8DI;
{attribute 'TcLinkTo' := '
.bIn1 := TIIB(73)^Channel 1^Input;
.bIn2 := TIIB(73)^Channel 2^Input;
.bIn3 := TIIB(73)^Channel 3^Input;
.bIn4 := TIIB(73)^Channel 4^Input;
.bIn5 := TIIB(73)^Channel 5^Input;
.bIn6 := TIIB(73)^Channel 6^Input;
.bIn7 := TIIB(73)^Channel 7^Input;
.bIn8 := TIIB(73)^Channel 8^Input'}
FG_01_EL1008_2 : ST_Beckhoff_8DI;
{attribute 'TcLinkTo' := '
.bOut1 := TIIB(74)^Channel 1^Output;
.bOut2 := TIIB(74)^Channel 2^Output;
.bOut3 := TIIB(74)^Channel 3^Output;
.bOut4 := TIIB(74)^Channel 4^Output;
.bOut5 := TIIB(74)^Channel 5^Output;
.bOut6 := TIIB(74)^Channel 6^Output;
.bOut7 := TIIB(74)^Channel 7^Output;
.bOut8 := TIIB(74)^Channel 8^Output'}
FG_01_EL2008_1 : ST_Beckhoff_8DO;
{attribute 'TcLinkTo' := '
.bIn1 := TIIB(75)^Channel 1^Input;
.bIn2 := TIIB(75)^Channel 2^Input;
.bIn3 := TIIB(75)^Channel 3^Input;
.bIn4 := TIIB(75)^Channel 4^Input;
.bIn5 := TIIB(75)^Channel 5^Input;
.bIn6 := TIIB(75)^Channel 6^Input;
.bIn7 := TIIB(75)^Channel 7^Input;
.bIn8 := TIIB(75)^Channel 8^Input;
.bOut1 := TIIB(75)^Channel 9^Output;
.bOut2 := TIIB(75)^Channel 10^Output;
.bOut3 := TIIB(75)^Channel 11^Output;
.bOut4 := TIIB(75)^Channel 12^Output;
.bOut5 := TIIB(75)^Channel 13^Output;
.bOut6 := TIIB(75)^Channel 14^Output;
.bOut7 := TIIB(75)^Channel 15^Output;
.bOut8 := TIIB(75)^Channel 16^Output'}
FG_01_EL1859_1 : ST_Beckhoff_8DI_8DO;
{attribute 'TcLinkTo' := '
.bIn1 := TIIB(76)^Channel 1^Input;
.bIn2 := TIIB(76)^Channel 2^Input;
.bIn3 := TIIB(76)^Channel 3^Input;
.bIn4 := TIIB(76)^Channel 4^Input;
.bIn5 := TIIB(76)^Channel 5^Input;
.bIn6 := TIIB(76)^Channel 6^Input;
.bIn7 := TIIB(76)^Channel 7^Input;
.bIn8 := TIIB(76)^Channel 8^Input;
.bOut1 := TIIB(76)^Channel 9^Output;
.bOut2 := TIIB(76)^Channel 10^Output;
.bOut3 := TIIB(76)^Channel 11^Output;
.bOut4 := TIIB(76)^Channel 12^Output;
.bOut5 := TIIB(76)^Channel 13^Output;
.bOut6 := TIIB(76)^Channel 14^Output;
.bOut7 := TIIB(76)^Channel 15^Output;
.bOut8 := TIIB(76)^Channel 16^Output'}
FG_01_EL1859_2 : ST_Beckhoff_8DI_8DO;
{attribute 'TcLinkTo' := '
.bIn1 := TIIB(78)^Channel 1^Input;
.bIn2 := TIIB(78)^Channel 2^Input;
.bIn3 := TIIB(78)^Channel 3^Input;
.bIn4 := TIIB(78)^Channel 4^Input;
.bIn5 := TIIB(78)^Channel 5^Input;
.bIn6 := TIIB(78)^Channel 6^Input;
.bIn7 := TIIB(78)^Channel 7^Input;
.bIn8 := TIIB(78)^Channel 8^Input;
.bOut1 := TIIB(78)^Channel 9^Output;
.bOut2 := TIIB(78)^Channel 10^Output;
.bOut3 := TIIB(78)^Channel 11^Output;
.bOut4 := TIIB(78)^Channel 12^Output;
.bOut5 := TIIB(78)^Channel 13^Output;
.bOut6 := TIIB(78)^Channel 14^Output;
.bOut7 := TIIB(78)^Channel 15^Output;
.bOut8 := TIIB(78)^Channel 16^Output'}
FG_02_EL1859_1 : ST_Beckhoff_8DI_8DO;
{attribute 'TcLinkTo' := '
.bIn1 := TIIB(80)^Channel 1^Input;
.bIn2 := TIIB(80)^Channel 2^Input;
.bIn3 := TIIB(80)^Channel 3^Input;
.bIn4 := TIIB(80)^Channel 4^Input;
.bIn5 := TIIB(80)^Channel 5^Input;
.bIn6 := TIIB(80)^Channel 6^Input;
.bIn7 := TIIB(80)^Channel 7^Input;
.bIn8 := TIIB(80)^Channel 8^Input;
.bIn9 := TIIB(80)^Channel 9^Input;
.bIn10 := TIIB(80)^Channel 10^Input;
.bIn11 := TIIB(80)^Channel 11^Input;
.bIn12 := TIIB(80)^Channel 12^Input;
.bIn13 := TIIB(80)^Channel 13^Input;
.bIn14 := TIIB(80)^Channel 14^Input;
.bIn15 := TIIB(80)^Channel 15^Input;
.bIn16 := TIIB(80)^Channel 16^Input'}
FG_03_EL1809_1 : ST_Beckhoff_16DI;
{attribute 'TcLinkTo' := '
.bOut1 := TIIB(81)^Channel 1^Output;
.bOut2 := TIIB(81)^Channel 2^Output;
.bOut3 := TIIB(81)^Channel 3^Output;
.bOut4 := TIIB(81)^Channel 4^Output;
.bOut5 := TIIB(81)^Channel 5^Output;
.bOut6 := TIIB(81)^Channel 6^Output;
.bOut7 := TIIB(81)^Channel 7^Output;
.bOut8 := TIIB(81)^Channel 8^Output;
.bOut9 := TIIB(81)^Channel 9^Output;
.bOut10 := TIIB(81)^Channel 10^Output;
.bOut11 := TIIB(81)^Channel 11^Output;
.bOut12 := TIIB(81)^Channel 12^Output;
.bOut13 := TIIB(81)^Channel 13^Output;
.bOut14 := TIIB(81)^Channel 14^Output;
.bOut15 := TIIB(81)^Channel 15^Output;
.bOut16 := TIIB(81)^Channel 16^Output'}
FG_03_EL2809_1 : ST_Beckhoff_16DO;
{attribute 'TcLinkTo' := '
.bIn1 := TIIB(83)^Channel 1^Input;
.bIn2 := TIIB(83)^Channel 2^Input;
.bIn3 := TIIB(83)^Channel 3^Input;
.bIn4 := TIIB(83)^Channel 4^Input;
.bIn5 := TIIB(83)^Channel 5^Input;
.bIn6 := TIIB(83)^Channel 6^Input;
.bIn7 := TIIB(83)^Channel 7^Input;
.bIn8 := TIIB(83)^Channel 8^Input'}
FG_04_EL1008_1 : ST_Beckhoff_8DI;
{attribute 'TcLinkTo' := '
.bOut1 := TIIB(84)^Channel 1^Output;
.bOut2 := TIIB(84)^Channel 2^Output;
.bOut3 := TIIB(84)^Channel 3^Output;
.bOut4 := TIIB(84)^Channel 4^Output;
.bOut5 := TIIB(84)^Channel 5^Output;
.bOut6 := TIIB(84)^Channel 6^Output;
.bOut7 := TIIB(84)^Channel 7^Output;
.bOut8 := TIIB(84)^Channel 8^Output'}
FG_04_EL2008_1 : ST_Beckhoff_8DO;
{attribute 'TcLinkTo' := '
.bIn1 := TIIB(86)^Channel 1^Input;
.bIn2 := TIIB(86)^Channel 2^Input;
.bIn3 := TIIB(86)^Channel 3^Input;
.bIn4 := TIIB(86)^Channel 4^Input;
.bIn5 := TIIB(86)^Channel 5^Input;
.bIn6 := TIIB(86)^Channel 6^Input;
.bIn7 := TIIB(86)^Channel 7^Input;
.bIn8 := TIIB(86)^Channel 8^Input;
.bIn9 := TIIB(86)^Channel 9^Input;
.bIn10 := TIIB(86)^Channel 10^Input;
.bIn11 := TIIB(86)^Channel 11^Input;
.bIn12 := TIIB(86)^Channel 12^Input;
.bIn13 := TIIB(86)^Channel 13^Input;
.bIn14 := TIIB(86)^Channel 14^Input;
.bIn15 := TIIB(86)^Channel 15^Input;
.bIn16 := TIIB(86)^Channel 16^Input'}
FG_05_EL1809_1 : ST_Beckhoff_16DI;
{attribute 'TcLinkTo' := '
.bOut1 := TIIB(87)^Channel 1^Output;
.bOut2 := TIIB(87)^Channel 2^Output;
.bOut3 := TIIB(87)^Channel 3^Output;
.bOut4 := TIIB(87)^Channel 4^Output;
.bOut5 := TIIB(87)^Channel 5^Output;
.bOut6 := TIIB(87)^Channel 6^Output;
.bOut7 := TIIB(87)^Channel 7^Output;
.bOut8 := TIIB(87)^Channel 8^Output;
.bOut9 := TIIB(87)^Channel 9^Output;
.bOut10 := TIIB(87)^Channel 10^Output;
.bOut11 := TIIB(87)^Channel 11^Output;
.bOut12 := TIIB(87)^Channel 12^Output;
.bOut13 := TIIB(87)^Channel 13^Output;
.bOut14 := TIIB(87)^Channel 14^Output;
.bOut15 := TIIB(87)^Channel 15^Output;
.bOut16 := TIIB(87)^Channel 16^Output'}
FG_05_EL2809_1 : ST_Beckhoff_16DO;
{attribute 'TcLinkTo' := '
.bIn1 := TIIB(88)^Channel 1^Input;
.bIn2 := TIIB(88)^Channel 2^Input;
.bIn3 := TIIB(88)^Channel 3^Input;
.bIn4 := TIIB(88)^Channel 4^Input;
.bIn5 := TIIB(88)^Channel 5^Input;
.bIn6 := TIIB(88)^Channel 6^Input;
.bIn7 := TIIB(88)^Channel 7^Input;
.bIn8 := TIIB(88)^Channel 8^Input;
.bOut1 := TIIB(88)^Channel 9^Output;
.bOut2 := TIIB(88)^Channel 10^Output;
.bOut3 := TIIB(88)^Channel 11^Output;
.bOut4 := TIIB(88)^Channel 12^Output;
.bOut5 := TIIB(88)^Channel 13^Output;
.bOut6 := TIIB(88)^Channel 14^Output;
.bOut7 := TIIB(88)^Channel 15^Output;
.bOut8 := TIIB(88)^Channel 16^Output'}
FG_05_EL1859_1 : ST_Beckhoff_8DI_8DO;
{attribute 'TcLinkTo' := '
.bIn1 := TIIB(89)^Channel 1^Input;
.bIn2 := TIIB(89)^Channel 2^Input;
.bIn3 := TIIB(89)^Channel 3^Input;
.bIn4 := TIIB(89)^Channel 4^Input;
.bIn5 := TIIB(89)^Channel 5^Input;
.bIn6 := TIIB(89)^Channel 6^Input;
.bIn7 := TIIB(89)^Channel 7^Input;
.bIn8 := TIIB(89)^Channel 8^Input;
.bOut1 := TIIB(89)^Channel 9^Output;
.bOut2 := TIIB(89)^Channel 10^Output;
.bOut3 := TIIB(89)^Channel 11^Output;
.bOut4 := TIIB(89)^Channel 12^Output;
.bOut5 := TIIB(89)^Channel 13^Output;
.bOut6 := TIIB(89)^Channel 14^Output;
.bOut7 := TIIB(89)^Channel 15^Output;
.bOut8 := TIIB(89)^Channel 16^Output'}
FG_05_EL1859_2 : ST_Beckhoff_8DI_8DO;
END_VAR

// ---- Hil/EtherCAT_1_SIM/PRG_EtherCAT_1_SIM.TcPOU
PROGRAM PRG_EtherCAT_1_SIM
VAR
END_VAR

END_PROGRAM

// ---- FG_01/FG_01.TcPOU
FUNCTION_BLOCK FG_01

{region generated code}
VAR_INPUT
	B_SafetyGate1 : FB_SensorBinary;
	B_SafetyGate2 : FB_SensorBinary;
	P_Camera : FB_Camera;
	Y_Gate1 : FB_Cylinder;
	Y_Gate2 : FB_Cylinder;
	Y_Gripper : FB_Cylinder;
	Y_LaserMark : FB_DeviceByte;
	Y_Platform : FB_Cylinder;
	Y_ReaderWindow : FB_Cylinder;
END_VAR
{endregion}

{region generated code}
	InitRun();
	B_SafetyGate1();
	B_SafetyGate2();
	P_Camera();
	Y_Gate1();
	Y_Gate2();
	Y_Gripper();
	Y_LaserMark();
	Y_Platform();
	Y_ReaderWindow();
{endregion}

Mapping();

METHOD InitRun
{region generated code}
VAR_INST
	bInitRun : BOOL := TRUE;
END_VAR
{endregion}
{region generated code}
	IF NOT bInitRun THEN RETURN; END_IF
	bInitRun := FALSE;
{endregion}
END_METHOD

ACTION Mapping:
// ============================================================================
// FG_01 twin <-> EtherCAT simulation process image.
//
// The discrete cylinders and sensors remain on the shared EL1008/EL2008 cards.
// Each byte device owns an EL1859, so its complete control and status bytes
// travel together instead of borrowing individual channels from those cards.
// GVL_EtherCAT_1_SIM is generated from the SIM master and carries the TIIB ids.
// ============================================================================

// --- Y_Gripper - double solenoid --------------------------------------------
// DI 1/2, DO 1/5. It was a single solenoid with a spring return and no retract
// coil at all; the control side is FB_DoubleSolenoidFeedback now, so the coil
// exists and has to be driven from here or the twin cylinder never leaves the
// extended limit once bExtend drops.
//
// THE PAIR IS NOT ADJACENT. The extend coil keeps DO 1 and the new retract coil
// took the lowest free output on the card, which is 5 - renumbering the four
// coils in between would have rewired FG_01 for cosmetics.
GVL_EtherCAT_1_SIM.FG_01_EL1008_1.bIn1	:= Y_Gripper.bRetracted;
GVL_EtherCAT_1_SIM.FG_01_EL1008_1.bIn2	:= Y_Gripper.bExtended;
Y_Gripper.bExtend		:= GVL_EtherCAT_1_SIM.FG_01_EL2008_1.bOut1;
Y_Gripper.bRetract		:= GVL_EtherCAT_1_SIM.FG_01_EL2008_1.bOut5;

// --- Y_Platform - double solenoid -------------------------------------------
// DI 3/4, DO 2/3.
GVL_EtherCAT_1_SIM.FG_01_EL1008_1.bIn3	:= Y_Platform.bRetracted;
GVL_EtherCAT_1_SIM.FG_01_EL1008_1.bIn4	:= Y_Platform.bExtended;
Y_Platform.bExtend		:= GVL_EtherCAT_1_SIM.FG_01_EL2008_1.bOut2;
Y_Platform.bRetract		:= GVL_EtherCAT_1_SIM.FG_01_EL2008_1.bOut3;

// --- Y_ReaderWindow - double solenoid ---------------------------------------
// DI 5/6, DO 4/6. Same change as Y_Gripper above, and the pair is split for the
// same reason: extend keeps DO 4, retract took the next free output.
GVL_EtherCAT_1_SIM.FG_01_EL1008_1.bIn5	:= Y_ReaderWindow.bRetracted;
GVL_EtherCAT_1_SIM.FG_01_EL1008_1.bIn6	:= Y_ReaderWindow.bExtended;
Y_ReaderWindow.bExtend	:= GVL_EtherCAT_1_SIM.FG_01_EL2008_1.bOut4;
Y_ReaderWindow.bRetract	:= GVL_EtherCAT_1_SIM.FG_01_EL2008_1.bOut6;

// --- P_Camera: FG_01_EL1859_1 ----------------------------------------------
// Was P_Reader, an FB_Reader whose whole byte was copied across because the byte
// was the interface. It is a camera now, with six named signals and four bits on
// the wire, and the bit positions below are the contract with FB_AbstractCamera
// in OC_PLC:
//
//   DO 1 (Ch 9)  Enable        DI 1 (Ch 1)  Ready
//   DO 2 (Ch 10) Trigger       DI 2 (Ch 2)  Busy
//                              DI 3 (Ch 3)  ResultValid
//                              DI 4 (Ch 4)  ResultOK
//
// The SIM box id is deliberately not written here. It used to say TIIB 45; the
// EtherCAT emulation was rebuilt, every box renumbered, and the comment became
// quietly wrong while the GVL it describes stayed correct. GVL_EtherCAT_1_SIM is
// regenerated with the emulation and is the only place that id belongs.

// What the part must be carrying. FG_01 is the identify station: the twin's
// DataReader reads the payload's SerialNumber key, and Assembly Part 1 carries
// 60. A pallet with no part, or a part with no serial number, reads 0 and fails.
//
// SET HERE AND NOT IN InitRun BECAUSE Mapping IS THE ONLY ACTION WE OWN - OC
// Assistant regenerates everything inside the {region generated code} blocks on
// the next twin regeneration.
P_Camera.nExpectedData := 60;

P_Camera.bEnable	:= GVL_EtherCAT_1_SIM.FG_01_EL1859_1.bOut1;
P_Camera.bTrigger	:= GVL_EtherCAT_1_SIM.FG_01_EL1859_1.bOut2;

GVL_EtherCAT_1_SIM.FG_01_EL1859_1.bIn1 := P_Camera.bReady;
GVL_EtherCAT_1_SIM.FG_01_EL1859_1.bIn2 := P_Camera.bBusy;
GVL_EtherCAT_1_SIM.FG_01_EL1859_1.bIn3 := P_Camera.bResultValid;
GVL_EtherCAT_1_SIM.FG_01_EL1859_1.bIn4 := P_Camera.bResultOK;

// --- Y_LaserMark: FG_01_EL1859_2 -------------------------------------------
// FB_DeviceByte stores its byte interface in the low eight bits of the data words.
Y_LaserMark.nControlData.0 := GVL_EtherCAT_1_SIM.FG_01_EL1859_2.bOut1;
Y_LaserMark.nControlData.1 := GVL_EtherCAT_1_SIM.FG_01_EL1859_2.bOut2;
Y_LaserMark.nControlData.2 := GVL_EtherCAT_1_SIM.FG_01_EL1859_2.bOut3;
Y_LaserMark.nControlData.3 := GVL_EtherCAT_1_SIM.FG_01_EL1859_2.bOut4;
Y_LaserMark.nControlData.4 := GVL_EtherCAT_1_SIM.FG_01_EL1859_2.bOut5;
Y_LaserMark.nControlData.5 := GVL_EtherCAT_1_SIM.FG_01_EL1859_2.bOut6;
Y_LaserMark.nControlData.6 := GVL_EtherCAT_1_SIM.FG_01_EL1859_2.bOut7;
Y_LaserMark.nControlData.7 := GVL_EtherCAT_1_SIM.FG_01_EL1859_2.bOut8;
GVL_EtherCAT_1_SIM.FG_01_EL1859_2.bIn1 := Y_LaserMark.nStatusData.0;
GVL_EtherCAT_1_SIM.FG_01_EL1859_2.bIn2 := Y_LaserMark.nStatusData.1;
GVL_EtherCAT_1_SIM.FG_01_EL1859_2.bIn3 := Y_LaserMark.nStatusData.2;
GVL_EtherCAT_1_SIM.FG_01_EL1859_2.bIn4 := Y_LaserMark.nStatusData.3;
GVL_EtherCAT_1_SIM.FG_01_EL1859_2.bIn5 := Y_LaserMark.nStatusData.4;
GVL_EtherCAT_1_SIM.FG_01_EL1859_2.bIn6 := Y_LaserMark.nStatusData.5;
GVL_EtherCAT_1_SIM.FG_01_EL1859_2.bIn7 := Y_LaserMark.nStatusData.6;
GVL_EtherCAT_1_SIM.FG_01_EL1859_2.bIn8 := Y_LaserMark.nStatusData.7;

// --- Y_Gate1 / Y_Gate2 - single solenoid, spring return ---------------------
// Moved in from FG_Transport with the twin. EXTEND CLOSES the gate; the spring
// opens it, so both limits are read and the coil is the closing command.
// EL1008 #2 DI 1..4, EL2008 #1 DO 7/8.
Y_Gate1.bExtend		:= GVL_EtherCAT_1_SIM.FG_01_EL2008_1.bOut7;
GVL_EtherCAT_1_SIM.FG_01_EL1008_2.bIn1	:= Y_Gate1.bRetracted;
GVL_EtherCAT_1_SIM.FG_01_EL1008_2.bIn2	:= Y_Gate1.bExtended;

Y_Gate2.bExtend		:= GVL_EtherCAT_1_SIM.FG_01_EL2008_1.bOut8;
GVL_EtherCAT_1_SIM.FG_01_EL1008_2.bIn3	:= Y_Gate2.bRetracted;
GVL_EtherCAT_1_SIM.FG_01_EL1008_2.bIn4	:= Y_Gate2.bExtended;

// --- B_SafetyGate1 / B_SafetyGate2 -----------------------------------------
// Independent gate position monitoring, moved across with the gates. The control
// side reads these through each FB_DigitalSensor's own HardwareInput, so they
// appear in no GVL - but the twin still has to drive the channels.
// EL1008 #2 DI 5/6.
GVL_EtherCAT_1_SIM.FG_01_EL1008_2.bIn5	:= B_SafetyGate1.bValue;
GVL_EtherCAT_1_SIM.FG_01_EL1008_2.bIn6	:= B_SafetyGate2.bValue;

// Spare after FG_01: EL1008 #1 DI 7/8; EL1008 #2 DI 7/8;
// EL1859 #1 DI 5..8 and DO 3..8, freed when P_Reader became P_Camera.
//
// EL2008 #1 IS NOW FULL. DO 5/6 were the last two free outputs on it and the
// Y_Gripper / Y_ReaderWindow retract coils took them. A further coil in this
// group needs another EL2008 on the FG_01 coupler, on both masters.
END_ACTION

END_FUNCTION_BLOCK

// ---- FG_02/FG_02.TcPOU
FUNCTION_BLOCK FG_02

{region generated code}
VAR_INPUT
	P_Camera : FB_Camera;
END_VAR
{endregion}

{region generated code}
	InitRun();
	P_Camera();
{endregion}

Mapping();

METHOD InitRun
{region generated code}
VAR_INST
	bInitRun : BOOL := TRUE;
END_VAR
{endregion}
{region generated code}
	IF NOT bInitRun THEN RETURN; END_IF
	bInitRun := FALSE;
{endregion}
END_METHOD

ACTION Mapping:
// ============================================================================
// FG_02 twin <-> EtherCAT simulation process image.
//
// One device, one card. P_Camera owns FG_02_EL1859_1 outright, so the whole
// interface travels together rather than borrowing bits from a shared card.
//
// THE BYTE IS NO LONGER COPIED WHOLESALE. It used to be, because the device was
// an FB_DeviceByte and the byte WAS the interface - a half-mapped byte would have
// been the thing that reads plausible and is wrong. FB_Camera is not a byte
// device: it exposes six named signals, and the bit positions below are the
// contract with FB_AbstractCamera in OC_PLC. Mapping bits 5..8 to nothing is
// correct now, because there is nothing on them.
//
//   DO 1 (Ch 9)  Enable        DI 1 (Ch 1)  Ready
//   DO 2 (Ch 10) Trigger       DI 2 (Ch 2)  Busy
//                              DI 3 (Ch 3)  ResultValid
//                              DI 4 (Ch 4)  ResultOK
//
// The GVL holds the SIM box id and is regenerated with the emulation, so it is
// deliberately not repeated here - that is what went stale in FG_01 when the
// emulation was rebuilt.
// ============================================================================

// --- P_Camera - what the part must be carrying ------------------------------
// FG_02 inspects the mark FG_01 applied: the laser writes LaserMark := 240 onto
// the payload, this station reads that key back and passes only on 240. A part
// that skipped FG_01, or whose mark failed, reads 0 and is a NOK.
//
// IT IS SET HERE AND NOT IN InitRun BECAUSE Mapping IS THE ONLY ACTION WE OWN -
// OC Assistant regenerates everything inside the {region generated code} blocks
// on the next twin regeneration.
P_Camera.nExpectedData := 240;

// --- P_Camera - the handshake on FG_02_EL1859_1 -----------------------------
// Commands from the control PLC.
P_Camera.bEnable	:= GVL_EtherCAT_1_SIM.FG_02_EL1859_1.bOut1;
P_Camera.bTrigger	:= GVL_EtherCAT_1_SIM.FG_02_EL1859_1.bOut2;

// The camera's answer. Ready, Busy and the verdict are synthesised inside
// FB_Camera - the Unity DataReader below it only echoes the two commands and
// hands over the datum it read.
GVL_EtherCAT_1_SIM.FG_02_EL1859_1.bIn1 := P_Camera.bReady;
GVL_EtherCAT_1_SIM.FG_02_EL1859_1.bIn2 := P_Camera.bBusy;
GVL_EtherCAT_1_SIM.FG_02_EL1859_1.bIn3 := P_Camera.bResultValid;
GVL_EtherCAT_1_SIM.FG_02_EL1859_1.bIn4 := P_Camera.bResultOK;

// Spare after FG_02: FG_02_EL1859_1 DI 5..8, DO 3..8.
END_ACTION

END_FUNCTION_BLOCK

// ---- FG_03/FG_03.TcPOU
FUNCTION_BLOCK FG_03

{region generated code}
VAR_INPUT
	B_Detect1 : FB_SensorBinary;
	B_Detect2 : FB_SensorBinary;
	Y_AxisR1 : FB_Cylinder;
	Y_AxisX1 : FB_Cylinder;
	Y_AxisX2 : FB_Cylinder;
	Y_AxisY1 : FB_Cylinder;
	Y_AxisY2 : FB_Cylinder;
	Y_Gripper1 : FB_Cylinder;
	Y_Gripper2 : FB_Cylinder;
END_VAR
{endregion}

{region generated code}
	InitRun();
	B_Detect1();
	B_Detect2();
	Y_AxisR1();
	Y_AxisX1();
	Y_AxisX2();
	Y_AxisY1();
	Y_AxisY2();
	Y_Gripper1();
	Y_Gripper2();
{endregion}

Mapping();

METHOD InitRun
{region generated code}
VAR_INST
	bInitRun : BOOL := TRUE;
END_VAR
{endregion}
{region generated code}
	IF NOT bInitRun THEN RETURN; END_IF
	bInitRun := FALSE;
{endregion}
END_METHOD

ACTION Mapping:
// ============================================================================
// FG_03 twin <-> EtherCAT simulation process image.
//
// Seven double solenoids and two grip sensors. Every solenoid gets two limit
// switches on FG_03_EL1809_1 and two coils on FG_03_EL2809_1, paired on matching
// channel numbers so a cylinder's DI n/n+1 and DO n/n+1 line up - which is what
// makes a wiring fault visible by inspection rather than by symptom.
//
// Channel order follows the process image, so EXTENDED IS THE LOW CHANNEL of each
// pair here. FG_01 has retracted first; neither is a convention, both are just
// what the allocator read off the declaration order.
//
// THE TWO SENSORS TAKE 15 AND 16, WHICH FILLS THE TERMINAL. B_Detect1 and B_Detect2
// are beam sensors inside the two grippers' jaws; they are inputs only, so they need
// no output channel and none is reserved for them. FG_03_EL1809_1 has no free input
// left after these two - the next input this group grows needs another card.
// ============================================================================

// --- Y_AxisR1 - double solenoid, both coils and both limits ----------------
// DI FG_03_EL1809_1 5/6, DO FG_03_EL2809_1 5/6.
GVL_EtherCAT_1_SIM.FG_03_EL1809_1.bIn5	:= Y_AxisR1.bExtended;
GVL_EtherCAT_1_SIM.FG_03_EL1809_1.bIn6	:= Y_AxisR1.bRetracted;
Y_AxisR1.bExtend	:= GVL_EtherCAT_1_SIM.FG_03_EL2809_1.bOut5;
Y_AxisR1.bRetract	:= GVL_EtherCAT_1_SIM.FG_03_EL2809_1.bOut6;

// --- Y_AxisX1 - double solenoid, both coils and both limits ----------------
// DI FG_03_EL1809_1 1/2, DO FG_03_EL2809_1 1/2.
GVL_EtherCAT_1_SIM.FG_03_EL1809_1.bIn1	:= Y_AxisX1.bExtended;
GVL_EtherCAT_1_SIM.FG_03_EL1809_1.bIn2	:= Y_AxisX1.bRetracted;
Y_AxisX1.bExtend	:= GVL_EtherCAT_1_SIM.FG_03_EL2809_1.bOut1;
Y_AxisX1.bRetract	:= GVL_EtherCAT_1_SIM.FG_03_EL2809_1.bOut2;

// --- Y_AxisX2 - double solenoid, both coils and both limits ----------------
// DI FG_03_EL1809_1 9/10, DO FG_03_EL2809_1 9/10.
GVL_EtherCAT_1_SIM.FG_03_EL1809_1.bIn9	:= Y_AxisX2.bExtended;
GVL_EtherCAT_1_SIM.FG_03_EL1809_1.bIn10	:= Y_AxisX2.bRetracted;
Y_AxisX2.bExtend	:= GVL_EtherCAT_1_SIM.FG_03_EL2809_1.bOut9;
Y_AxisX2.bRetract	:= GVL_EtherCAT_1_SIM.FG_03_EL2809_1.bOut10;

// --- Y_AxisY1 - double solenoid, both coils and both limits ----------------
// DI FG_03_EL1809_1 3/4, DO FG_03_EL2809_1 3/4.
GVL_EtherCAT_1_SIM.FG_03_EL1809_1.bIn3	:= Y_AxisY1.bExtended;
GVL_EtherCAT_1_SIM.FG_03_EL1809_1.bIn4	:= Y_AxisY1.bRetracted;
Y_AxisY1.bExtend	:= GVL_EtherCAT_1_SIM.FG_03_EL2809_1.bOut3;
Y_AxisY1.bRetract	:= GVL_EtherCAT_1_SIM.FG_03_EL2809_1.bOut4;

// --- Y_AxisY2 - double solenoid, both coils and both limits ----------------
// DI FG_03_EL1809_1 11/12, DO FG_03_EL2809_1 11/12.
GVL_EtherCAT_1_SIM.FG_03_EL1809_1.bIn11	:= Y_AxisY2.bExtended;
GVL_EtherCAT_1_SIM.FG_03_EL1809_1.bIn12	:= Y_AxisY2.bRetracted;
Y_AxisY2.bExtend	:= GVL_EtherCAT_1_SIM.FG_03_EL2809_1.bOut11;
Y_AxisY2.bRetract	:= GVL_EtherCAT_1_SIM.FG_03_EL2809_1.bOut12;

// --- Y_Gripper1 - double solenoid, both coils and both limits --------------
// DI FG_03_EL1809_1 7/8, DO FG_03_EL2809_1 7/8.
GVL_EtherCAT_1_SIM.FG_03_EL1809_1.bIn7	:= Y_Gripper1.bExtended;
GVL_EtherCAT_1_SIM.FG_03_EL1809_1.bIn8	:= Y_Gripper1.bRetracted;
Y_Gripper1.bExtend	:= GVL_EtherCAT_1_SIM.FG_03_EL2809_1.bOut7;
Y_Gripper1.bRetract	:= GVL_EtherCAT_1_SIM.FG_03_EL2809_1.bOut8;

// --- Y_Gripper2 - double solenoid, both coils and both limits --------------
// DI FG_03_EL1809_1 13/14, DO FG_03_EL2809_1 13/14.
GVL_EtherCAT_1_SIM.FG_03_EL1809_1.bIn13	:= Y_Gripper2.bExtended;
GVL_EtherCAT_1_SIM.FG_03_EL1809_1.bIn14	:= Y_Gripper2.bRetracted;
Y_Gripper2.bExtend	:= GVL_EtherCAT_1_SIM.FG_03_EL2809_1.bOut13;
Y_Gripper2.bRetract	:= GVL_EtherCAT_1_SIM.FG_03_EL2809_1.bOut14;

// --- B_Detect1 - part in the jaws of gripper 1, input only -----------------
// DI FG_03_EL1809_1 15. It follows its gripper's channel pair (7/8) in meaning but
// not in number: the pairs were allocated before these sensors existed, so the two
// of them take what was left at the end of the terminal.
GVL_EtherCAT_1_SIM.FG_03_EL1809_1.bIn15	:= B_Detect1.bValue;

// --- B_Detect2 - part in the jaws of gripper 2, input only -----------------
// DI FG_03_EL1809_1 16. The terminal is full after this one.
GVL_EtherCAT_1_SIM.FG_03_EL1809_1.bIn16	:= B_Detect2.bValue;
END_ACTION

END_FUNCTION_BLOCK

// ---- FG_04/FG_04.TcPOU
FUNCTION_BLOCK FG_04
{region generated code}
VAR_INPUT
	B_NIO : FB_SensorBinary;
	Y_AxisZ : FB_Cylinder;
END_VAR
{endregion}

{region generated code}
	InitRun();
	B_NIO();
	Y_AxisZ();
{endregion}

Mapping();

METHOD InitRun
{region generated code}
VAR_INST
	bInitRun : BOOL := TRUE;
END_VAR
{endregion}
{region generated code}
	IF NOT bInitRun THEN RETURN; END_IF
	bInitRun := FALSE;
{endregion}
END_METHOD

ACTION Mapping:
// ============================================================================
// FG_04 twin <-> EtherCAT simulation process image.
//
// The press and its verdict. Y_AxisZ is a double solenoid so that an abort
// mid-stroke leaves it where it is instead of letting a spring drive it further
// into the part.
//
// B_NIO is not a sensor reading. The twin's seating sensor is not a PLC symbol at
// all - its Link is disabled and it feeds PartPressDetector inside Unity, which
// publishes the conclusion here as one bit. The PLC reads it only at the bottom of
// the stroke with the hold expired.
// ============================================================================

// --- B_NIO - binary sensor -------------------------------------------------
// DI FG_04_EL1008_1 3.
GVL_EtherCAT_1_SIM.FG_04_EL1008_1.bIn3	:= B_NIO.bValue;

// --- Y_AxisZ - double solenoid, both coils and both limits -----------------
// DI FG_04_EL1008_1 1/2, DO FG_04_EL2008_1 1/2.
GVL_EtherCAT_1_SIM.FG_04_EL1008_1.bIn1	:= Y_AxisZ.bExtended;
GVL_EtherCAT_1_SIM.FG_04_EL1008_1.bIn2	:= Y_AxisZ.bRetracted;
Y_AxisZ.bExtend	:= GVL_EtherCAT_1_SIM.FG_04_EL2008_1.bOut1;
Y_AxisZ.bRetract	:= GVL_EtherCAT_1_SIM.FG_04_EL2008_1.bOut2;
END_ACTION

END_FUNCTION_BLOCK

// ---- FG_05/FG_05.TcPOU
FUNCTION_BLOCK FG_05

{region generated code}
VAR_INPUT
	B_Detect : FB_SensorBinary;
	B_Part : FB_SensorBinary;
	P_Camera : FB_Camera;
	Y_AxisR : FB_Cylinder;
	Y_AxisX : FB_Cylinder;
	Y_AxisZ1 : FB_Cylinder;
	Y_AxisZ2 : FB_Cylinder;
	Y_CapsSource : FB_DeviceByte;
	Y_CapsSourceStopper : FB_Cylinder;
	Y_Gripper : FB_Cylinder;
END_VAR
{endregion}

{region generated code}
	InitRun();
	B_Detect();
	B_Part();
	P_Camera();
	Y_AxisR();
	Y_AxisX();
	Y_AxisZ1();
	Y_AxisZ2();
	Y_CapsSource();
	Y_CapsSourceStopper();
	Y_Gripper();
{endregion}

Mapping();

METHOD InitRun
{region generated code}
VAR_INST
	bInitRun : BOOL := TRUE;
END_VAR
{endregion}
{region generated code}
	IF NOT bInitRun THEN RETURN; END_IF
	bInitRun := FALSE;
{endregion}
END_METHOD

ACTION Mapping:
// ============================================================================
// FG_05 twin <-> EtherCAT simulation process image.
//
// Six double solenoids, B_Part and B_Detect share FG_05_EL1809_1 /
// FG_05_EL2809_1. The two byte devices get a card each, as FG_01's do:
//
//   Y_CapsSource  FB_DeviceByte  FG_05_EL1859_1   control 0 table, 1 conveyor
//   P_Camera      FB_Camera      FG_05_EL1859_2   2 DO / 4 DI, see below
//
// The bunker reports nothing back, so its status byte is mapped and always reads
// zero. That is the honest wiring: the channels exist because the twin device is
// an FB_DeviceByte and carries nStatusData whatever this side does.
// ============================================================================

// --- B_Part - cap present at the pick position, on the FEED ----------------
// DI FG_05_EL1809_1 13.
GVL_EtherCAT_1_SIM.FG_05_EL1809_1.bIn13	:= B_Part.bValue;

// --- B_Detect - cap held in the gripper's JAWS, input only -----------------
// DI FG_05_EL1809_1 14. Not the same question as B_Part and not interchangeable
// with it: B_Part is on the feed and reports the next cap as soon as this one is
// lifted away. See the FG_05 block header in OC_PLC. Channels 15 and 16 stay free.
GVL_EtherCAT_1_SIM.FG_05_EL1809_1.bIn14	:= B_Detect.bValue;

// --- P_Camera: FG_05_EL1859_2 ----------------------------------------------
// Was an FB_Reader whose whole byte was copied across because the byte was the
// interface. It is a camera now - the third and last of the three optical devices
// to move - with six named signals and four bits on the wire. The bit positions
// are the contract with FB_AbstractCamera in OC_PLC and are IDENTICAL in FG_01,
// FG_02 and FG_05:
//
//   DO 1 (Ch 9)  Enable        DI 1 (Ch 1)  Ready
//   DO 2 (Ch 10) Trigger       DI 2 (Ch 2)  Busy
//                              DI 3 (Ch 3)  ResultValid
//                              DI 4 (Ch 4)  ResultOK
//
// The GVL holds the SIM box id and is regenerated with the emulation, so it is
// deliberately not repeated in this comment - that is what went stale in FG_01
// when the emulation was rebuilt.

// What the read has to return.
//
// IT READS THE ASSEMBLY ON THE PALLET, NOT THE CAP. The camera is mounted on the
// feed side but looks across at the pallet, and the key it reads - CapsID - is
// authored on Assembly Part 1, which carries 810. So the read answers "which cap
// does this assembly want", and the station passes only on the type it is set up
// to fit. An empty pallet reads 0 and fails.
//
// That is also why the read can sit before the pick: the pallet is already
// stopped and lifted by Index05 before FG_05 is triggered at all, so the assembly
// is in view from the first scan of the cycle.
//
// SET HERE AND NOT IN InitRun BECAUSE Mapping IS THE ONLY ACTION WE OWN - OC
// Assistant regenerates everything inside the {region generated code} blocks on
// the next twin regeneration.
P_Camera.nExpectedData := 810;

P_Camera.bEnable	:= GVL_EtherCAT_1_SIM.FG_05_EL1859_2.bOut1;
P_Camera.bTrigger	:= GVL_EtherCAT_1_SIM.FG_05_EL1859_2.bOut2;

GVL_EtherCAT_1_SIM.FG_05_EL1859_2.bIn1 := P_Camera.bReady;
GVL_EtherCAT_1_SIM.FG_05_EL1859_2.bIn2 := P_Camera.bBusy;
GVL_EtherCAT_1_SIM.FG_05_EL1859_2.bIn3 := P_Camera.bResultValid;
GVL_EtherCAT_1_SIM.FG_05_EL1859_2.bIn4 := P_Camera.bResultOK;

// --- Y_AxisR - double solenoid, both coils and both limits -----------------
// DI FG_05_EL1809_1 7/8, DO FG_05_EL2809_1 7/8.
GVL_EtherCAT_1_SIM.FG_05_EL1809_1.bIn7	:= Y_AxisR.bExtended;
GVL_EtherCAT_1_SIM.FG_05_EL1809_1.bIn8	:= Y_AxisR.bRetracted;
Y_AxisR.bExtend	:= GVL_EtherCAT_1_SIM.FG_05_EL2809_1.bOut7;
Y_AxisR.bRetract	:= GVL_EtherCAT_1_SIM.FG_05_EL2809_1.bOut8;

// --- Y_AxisX - double solenoid, both coils and both limits -----------------
// DI FG_05_EL1809_1 1/2, DO FG_05_EL2809_1 1/2.
GVL_EtherCAT_1_SIM.FG_05_EL1809_1.bIn1	:= Y_AxisX.bExtended;
GVL_EtherCAT_1_SIM.FG_05_EL1809_1.bIn2	:= Y_AxisX.bRetracted;
Y_AxisX.bExtend	:= GVL_EtherCAT_1_SIM.FG_05_EL2809_1.bOut1;
Y_AxisX.bRetract	:= GVL_EtherCAT_1_SIM.FG_05_EL2809_1.bOut2;

// --- Y_AxisZ1 - double solenoid, both coils and both limits ----------------
// DI FG_05_EL1809_1 3/4, DO FG_05_EL2809_1 3/4.
GVL_EtherCAT_1_SIM.FG_05_EL1809_1.bIn3	:= Y_AxisZ1.bExtended;
GVL_EtherCAT_1_SIM.FG_05_EL1809_1.bIn4	:= Y_AxisZ1.bRetracted;
Y_AxisZ1.bExtend	:= GVL_EtherCAT_1_SIM.FG_05_EL2809_1.bOut3;
Y_AxisZ1.bRetract	:= GVL_EtherCAT_1_SIM.FG_05_EL2809_1.bOut4;

// --- Y_AxisZ2 - double solenoid, both coils and both limits ----------------
// DI FG_05_EL1809_1 5/6, DO FG_05_EL2809_1 5/6.
GVL_EtherCAT_1_SIM.FG_05_EL1809_1.bIn5	:= Y_AxisZ2.bExtended;
GVL_EtherCAT_1_SIM.FG_05_EL1809_1.bIn6	:= Y_AxisZ2.bRetracted;
Y_AxisZ2.bExtend	:= GVL_EtherCAT_1_SIM.FG_05_EL2809_1.bOut5;
Y_AxisZ2.bRetract	:= GVL_EtherCAT_1_SIM.FG_05_EL2809_1.bOut6;

// --- Y_CapsSource - byte device, owns FG_05_EL1859_1 -----------------------
// Control byte PLC -> twin, status byte twin -> PLC. The card carries both,
// so the whole interface travels together instead of borrowing channels.
// The GVL holds the SIM box id and is regenerated with the emulation, so it
// is deliberately not repeated in this comment - that is what went stale in
// FG_01 when the emulation was rebuilt.
Y_CapsSource.nControlData.0 := GVL_EtherCAT_1_SIM.FG_05_EL1859_1.bOut1;
Y_CapsSource.nControlData.1 := GVL_EtherCAT_1_SIM.FG_05_EL1859_1.bOut2;
Y_CapsSource.nControlData.2 := GVL_EtherCAT_1_SIM.FG_05_EL1859_1.bOut3;
Y_CapsSource.nControlData.3 := GVL_EtherCAT_1_SIM.FG_05_EL1859_1.bOut4;
Y_CapsSource.nControlData.4 := GVL_EtherCAT_1_SIM.FG_05_EL1859_1.bOut5;
Y_CapsSource.nControlData.5 := GVL_EtherCAT_1_SIM.FG_05_EL1859_1.bOut6;
Y_CapsSource.nControlData.6 := GVL_EtherCAT_1_SIM.FG_05_EL1859_1.bOut7;
Y_CapsSource.nControlData.7 := GVL_EtherCAT_1_SIM.FG_05_EL1859_1.bOut8;
GVL_EtherCAT_1_SIM.FG_05_EL1859_1.bIn1 := Y_CapsSource.nStatusData.0;
GVL_EtherCAT_1_SIM.FG_05_EL1859_1.bIn2 := Y_CapsSource.nStatusData.1;
GVL_EtherCAT_1_SIM.FG_05_EL1859_1.bIn3 := Y_CapsSource.nStatusData.2;
GVL_EtherCAT_1_SIM.FG_05_EL1859_1.bIn4 := Y_CapsSource.nStatusData.3;
GVL_EtherCAT_1_SIM.FG_05_EL1859_1.bIn5 := Y_CapsSource.nStatusData.4;
GVL_EtherCAT_1_SIM.FG_05_EL1859_1.bIn6 := Y_CapsSource.nStatusData.5;
GVL_EtherCAT_1_SIM.FG_05_EL1859_1.bIn7 := Y_CapsSource.nStatusData.6;
GVL_EtherCAT_1_SIM.FG_05_EL1859_1.bIn8 := Y_CapsSource.nStatusData.7;

// --- Y_CapsSourceStopper - double solenoid, both coils and both limits -----
// DI FG_05_EL1809_1 11/12, DO FG_05_EL2809_1 11/12.
GVL_EtherCAT_1_SIM.FG_05_EL1809_1.bIn11	:= Y_CapsSourceStopper.bExtended;
GVL_EtherCAT_1_SIM.FG_05_EL1809_1.bIn12	:= Y_CapsSourceStopper.bRetracted;
Y_CapsSourceStopper.bExtend	:= GVL_EtherCAT_1_SIM.FG_05_EL2809_1.bOut11;
Y_CapsSourceStopper.bRetract	:= GVL_EtherCAT_1_SIM.FG_05_EL2809_1.bOut12;

// --- Y_Gripper - double solenoid, both coils and both limits ---------------
// DI FG_05_EL1809_1 9/10, DO FG_05_EL2809_1 9/10.
GVL_EtherCAT_1_SIM.FG_05_EL1809_1.bIn9	:= Y_Gripper.bExtended;
GVL_EtherCAT_1_SIM.FG_05_EL1809_1.bIn10	:= Y_Gripper.bRetracted;
Y_Gripper.bExtend	:= GVL_EtherCAT_1_SIM.FG_05_EL2809_1.bOut9;
Y_Gripper.bRetract	:= GVL_EtherCAT_1_SIM.FG_05_EL2809_1.bOut10;
END_ACTION

END_FUNCTION_BLOCK

// ---- FG_System/FG_System.TcPOU
FUNCTION_BLOCK FG_System

{region generated code}
VAR_INPUT
	B_SafetyDoor11 : FB_Lock;
	B_SafetyDoor12 : FB_Lock;
	B_SafetyDoor13 : FB_Lock;
	B_SafetyDoor21 : FB_Lock;
	B_SafetyDoor22 : FB_Lock;
	B_SafetyDoor23 : FB_Lock;
	H_ControlPanel : FB_Panel;
	H_SignalTower : FB_Panel;
	SS_EStop1 : FB_Button;
	SS_EStop2 : FB_Button;
END_VAR
{endregion}

{region generated code}
	InitRun();
	B_SafetyDoor11();
	B_SafetyDoor12();
	B_SafetyDoor13();
	B_SafetyDoor21();
	B_SafetyDoor22();
	B_SafetyDoor23();
	H_ControlPanel();
	H_SignalTower();
	SS_EStop1();
	SS_EStop2();
{endregion}

Mapping();

METHOD InitRun
{region generated code}
VAR_INST
	bInitRun : BOOL := TRUE;
END_VAR
{endregion}
{region generated code}
	IF NOT bInitRun THEN RETURN; END_IF
	bInitRun := FALSE;
{endregion}
END_METHOD

ACTION Mapping:
// ============================================================================
// FG_System twin <-> EtherCAT simulation process image.
//
// Mirrors Mapping_PLC.xml channel for channel. Panel channel order follows the
// twin's own PanelSampler bit order, verified 2026-08-20 against the live scene,
// so DI channel n and DO channel n are the same button and nothing here needs a
// lookup table:
//   H_ControlPanel  bit0 START  1 RESET  2 STOP   3 CLEAR
//                   bit4 ABORT  5 PRODUCTION  6 MAINTANANCE  7 MANUAL
//   H_SignalTower   bit0 RED    1 YELLOW  2 BLUE  3 GREEN
//
// Direction is baked into which side of the assignment the GVL sits on:
//   twin status  -> bIn*   the PLC reads it
//   bOut*        -> twin control   the PLC drives it
// ============================================================================

// --- H_ControlPanel buttons -> Panel DI 1..8 --------------------------------
// FB_Panel aggregates all eight buttons into one DWORD; the PLC sees eight
// separate channels, which is what lets FB_ControlSource's own located
// StartPressed / StopPressed / ResetPressed inputs link directly.
GVL_EtherCAT_1_SIM.FG_System_Panel_EL1809_1.bIn1	:= H_ControlPanel.nStatusData.0;	// START
GVL_EtherCAT_1_SIM.FG_System_Panel_EL1809_1.bIn2	:= H_ControlPanel.nStatusData.1;	// RESET
GVL_EtherCAT_1_SIM.FG_System_Panel_EL1809_1.bIn3	:= H_ControlPanel.nStatusData.2;	// STOP
GVL_EtherCAT_1_SIM.FG_System_Panel_EL1809_1.bIn4	:= H_ControlPanel.nStatusData.3;	// CLEAR
GVL_EtherCAT_1_SIM.FG_System_Panel_EL1809_1.bIn5	:= H_ControlPanel.nStatusData.4;	// ABORT
GVL_EtherCAT_1_SIM.FG_System_Panel_EL1809_1.bIn6	:= H_ControlPanel.nStatusData.5;	// PRODUCTION
GVL_EtherCAT_1_SIM.FG_System_Panel_EL1809_1.bIn7	:= H_ControlPanel.nStatusData.6;	// MAINTANANCE
GVL_EtherCAT_1_SIM.FG_System_Panel_EL1809_1.bIn8	:= H_ControlPanel.nStatusData.7;	// MANUAL

// --- Emergency stops -> Panel DI 9/10 ---------------------------------------
// FB_Button reports bValue TRUE while PRESSED, and these are Toggle type so a
// click latches. NOT is what makes the twin read like a real NC mushroom -
// TRUE while healthy, FALSE while latched - so PLC_1 needs no twin-only variant:
// FG_System.Initialize sets SS_EStop*.Inverted := TRUE for both cases.
// Do not drop the NOT without clearing that too, in the same edit.
// See _workflow/reference/plc-io-exceptions.md.
GVL_EtherCAT_1_SIM.FG_System_Panel_EL1809_1.bIn9	:= NOT SS_EStop1.bValue;
GVL_EtherCAT_1_SIM.FG_System_Panel_EL1809_1.bIn10	:= NOT SS_EStop2.bValue;

// --- Safety doors -> Door DI 1..12 ------------------------------------------
// Two channels per door, closed then locked, in twin order 11/12/13 then
// 21/22/23. Both are needed: closed alone does not make a guard secure.
GVL_EtherCAT_1_SIM.FG_System_Door_EL1809_1.bIn1		:= B_SafetyDoor11.bClosed;
GVL_EtherCAT_1_SIM.FG_System_Door_EL1809_1.bIn2		:= B_SafetyDoor11.bLocked;
GVL_EtherCAT_1_SIM.FG_System_Door_EL1809_1.bIn3		:= B_SafetyDoor12.bClosed;
GVL_EtherCAT_1_SIM.FG_System_Door_EL1809_1.bIn4		:= B_SafetyDoor12.bLocked;
GVL_EtherCAT_1_SIM.FG_System_Door_EL1809_1.bIn5		:= B_SafetyDoor13.bClosed;
GVL_EtherCAT_1_SIM.FG_System_Door_EL1809_1.bIn6		:= B_SafetyDoor13.bLocked;
GVL_EtherCAT_1_SIM.FG_System_Door_EL1809_1.bIn7		:= B_SafetyDoor21.bClosed;
GVL_EtherCAT_1_SIM.FG_System_Door_EL1809_1.bIn8		:= B_SafetyDoor21.bLocked;
GVL_EtherCAT_1_SIM.FG_System_Door_EL1809_1.bIn9		:= B_SafetyDoor22.bClosed;
GVL_EtherCAT_1_SIM.FG_System_Door_EL1809_1.bIn10	:= B_SafetyDoor22.bLocked;
GVL_EtherCAT_1_SIM.FG_System_Door_EL1809_1.bIn11	:= B_SafetyDoor23.bClosed;
GVL_EtherCAT_1_SIM.FG_System_Door_EL1809_1.bIn12	:= B_SafetyDoor23.bLocked;

// --- Panel DO 1..8 -> H_ControlPanel button lamps ---------------------------
// Same bit order as the buttons above, so channel n lights the button that
// channel n reads.
H_ControlPanel.nControlData.0	:= GVL_EtherCAT_1_SIM.FG_System_Panel_EL2809_1.bOut1;	// START
H_ControlPanel.nControlData.1	:= GVL_EtherCAT_1_SIM.FG_System_Panel_EL2809_1.bOut2;	// RESET
H_ControlPanel.nControlData.2	:= GVL_EtherCAT_1_SIM.FG_System_Panel_EL2809_1.bOut3;	// STOP
H_ControlPanel.nControlData.3	:= GVL_EtherCAT_1_SIM.FG_System_Panel_EL2809_1.bOut4;	// CLEAR
H_ControlPanel.nControlData.4	:= GVL_EtherCAT_1_SIM.FG_System_Panel_EL2809_1.bOut5;	// ABORT
H_ControlPanel.nControlData.5	:= GVL_EtherCAT_1_SIM.FG_System_Panel_EL2809_1.bOut6;	// PRODUCTION
H_ControlPanel.nControlData.6	:= GVL_EtherCAT_1_SIM.FG_System_Panel_EL2809_1.bOut7;	// MAINTANANCE
H_ControlPanel.nControlData.7	:= GVL_EtherCAT_1_SIM.FG_System_Panel_EL2809_1.bOut8;	// MANUAL

// --- Panel DO 9..12 -> H_SignalTower ----------------------------------------
// NOTE the tower is four lamps and GREEN is bit 3, not bit 2. The twin's
// authored prose said three lamps with GREEN at bit 2 until 2026-08-20.
H_SignalTower.nControlData.0	:= GVL_EtherCAT_1_SIM.FG_System_Panel_EL2809_1.bOut9;	// RED
H_SignalTower.nControlData.1	:= GVL_EtherCAT_1_SIM.FG_System_Panel_EL2809_1.bOut10;	// YELLOW
H_SignalTower.nControlData.2	:= GVL_EtherCAT_1_SIM.FG_System_Panel_EL2809_1.bOut11;	// BLUE
H_SignalTower.nControlData.3	:= GVL_EtherCAT_1_SIM.FG_System_Panel_EL2809_1.bOut12;	// GREEN

// --- Panel DO 13/14 -> the mushrooms' own lamps -----------------------------
// FB_Button.bEnable is the lamp: 0 off, 1 on, confirmed in the OC_Core binary.
// The twin's Emergency Switch prefab has _localFeedback FALSE, so these lamps
// light only because the PLC drives them - solid while latched, flashing while
// latched during Clearing.
SS_EStop1.bEnable	:= GVL_EtherCAT_1_SIM.FG_System_Panel_EL2809_1.bOut13;
SS_EStop2.bEnable	:= GVL_EtherCAT_1_SIM.FG_System_Panel_EL2809_1.bOut14;

// --- Door DO 1..6 -> the six safety locks -----------------------------------
// The PLC commands these locked throughout Production and releases them in
// Maintenance and Manual, which is the only way into the cell.
B_SafetyDoor11.bLock	:= GVL_EtherCAT_1_SIM.FG_System_Door_EL2008_1.bOut1;
B_SafetyDoor12.bLock	:= GVL_EtherCAT_1_SIM.FG_System_Door_EL2008_1.bOut2;
B_SafetyDoor13.bLock	:= GVL_EtherCAT_1_SIM.FG_System_Door_EL2008_1.bOut3;
B_SafetyDoor21.bLock	:= GVL_EtherCAT_1_SIM.FG_System_Door_EL2008_1.bOut4;
B_SafetyDoor22.bLock	:= GVL_EtherCAT_1_SIM.FG_System_Door_EL2008_1.bOut5;
B_SafetyDoor23.bLock	:= GVL_EtherCAT_1_SIM.FG_System_Door_EL2008_1.bOut6;

// Spare after FG_System: Panel EL1809 DI 11-16; Door EL1809 DI 13-16;
// Panel EL2809 DO 15-16; Door EL2008 DO 7-8.
END_ACTION

